// TwinCAT 3 PLC project XTS_PLC
// ProgramVersion: 3.1.4023.0
// libraries:
//   CmpBitmapPool, * (System)
//   Tc2_Math, * (Beckhoff Automation GmbH)
//   Tc2_MC2, * (Beckhoff Automation GmbH)
//   Tc2_Standard, * (Beckhoff Automation GmbH)
//   Tc2_System, * (Beckhoff Automation GmbH)
//   Tc2_Utilities, * (Beckhoff Automation GmbH)
//   Tc3_Mc3Definitions, * (Beckhoff Automation GmbH)
//   Tc3_McCollisionAvoidance, * (Beckhoff Automation GmbH)
//   Tc3_McCoordinatedMotion, * (Beckhoff Automation GmbH)
//   Tc3_Module, * (Beckhoff Automation GmbH)
//   Tc3_XTS_Utility, * (Beckhoff Automation GmbH)
//   VisuDialogs, * (System)
// project tree:
//   DUTs/ eColors.TcDUT, stFeedback.TcDUT, stStationCfg.TcDUT, stTableStructx10.TcDUT, stXTSCfg.TcDUT
//   / GlobalTextList.TcGTLO, PlcTask.TcTTO (not stored), VisualizationManager.TcVMO (not stored)
//   POUs/ MAIN.TcPOU, XTS_PRG.TcPOU
//   POUs/XTS/Group CA/ FB_GroupCA.TcPOU, VI_GroupCAVisu.TcVIS
//   POUs/XTS/Movers/ FB_Mover.TcPOU, FB_MoversFIFO.TcPOU (not stored), MC_JogCA.TcPOU, MC_MoveAbsoluteTimeCA.TcPOU, VI_MoverVisu.TcVIS, VI_MoversVisu.TcVIS
//   POUs/XTS/Stations/ FB_Station.TcPOU, VI_StationVISU.TcVIS, VI_StationsVISU.TcVIS
//   POUs/XTS/VISUs/ GlobalTextList_2.TcGTLO (not stored), VI_PLCOpenState.TcVIS, VI_XTSManualVisu.TcVIS, VI_XTSMainVisu.TcVIS, VI_XTSRunTimeVisu.TcVIS, VI_XTSConfigurationVisu.TcVIS, VI_XTSAutoVisu.TcVIS
//   POUs/XTS/VISUs/TextList/ AxisState_txt.TcTLO, GroupState_txt.TcTLO, MoverMode_TXT.TcTLO (not stored), MoversMode_txt.TcTLO, PML_Modes_txt.TcTLO, StationAckMode_txt.TcTLO (not stored)
//   POUs/XTS/ XTS_System.TcPOU
//   VISUs/ ImagePool.TcIPO (not stored), MAIN_VISU.TcVIS
// real-time tasks:
//   TASK XTS Task 1: cycle T#250us, priority 1, ADS port 350
//   TASK PlcTask: cycle T#10ms, priority 20, ADS port 351
//   TASK VISU_TASK: cycle T#50000us, priority 30, ADS port 352
//   TASK Job Task: cycle default, priority 32
//   TASK VISU_TASK1: cycle T#200000us, priority 2, ADS port 353
// motion (NC):
//   TASK NC-Task 1 SAF: cycle T#2ms, priority 4, ADS port 501
//   TASK NC-Task 1 SVB: cycle T#10ms, priority 8, ADS port 511
//   AXIS Mover Axis 1 (id 1)
//     Dynamic: AccelerationMaximum=80000, DecelerationMaximum=80000, Acceleration=20000, Deceleration=20000, Jerk=200000
//     Velo: Maximum=4000
//     PositionAreaControl: Enable=false
//     TargetPosControl: Enable=false
//     OtherSettings: AllowMotionCmdToSlave=true, AllowMotionCmdToExtSetGenAxis=true
//     encoder EncType=28
//       EncPara: ModuloFactor=10000, ToleranceWndModuloStart=0.2, Inverse=true, MaxCount=#xffffffff
//     drive DrvType=22
//       DrvPara: MaxCount=#xffffffff, DriveControlDWord=#x00000100
//         Analog: VeloReferenz=4200, TorqueSetpointScale=10
//         TimeComp: TaskDelayCycles=1
//     controller CtrType=1
//       CtrPara: PriorControlFactor=1
//         PosDiffControl: Range=10
//         Observer: BandWidth=20
//   AXIS Mover Axis 2 (id 2)
//     Dynamic: AccelerationMaximum=80000, DecelerationMaximum=80000, Acceleration=20000, Deceleration=20000, Jerk=200000
//     Velo: Maximum=4000
//     PositionAreaControl: Enable=false
//     TargetPosControl: Enable=false
//     OtherSettings: AllowMotionCmdToSlave=true, AllowMotionCmdToExtSetGenAxis=true
//     encoder EncType=28
//       EncPara: ModuloFactor=10000, ToleranceWndModuloStart=0.2, MaxCount=#xffffffff
//     drive DrvType=22
//       DrvPara: MaxCount=#xffffffff, DriveControlDWord=#x00000100
//         Analog: VeloReferenz=4200, TorqueSetpointScale=10
//         TimeComp: TaskDelayCycles=1
//     controller CtrType=1
//       CtrPara: PriorControlFactor=1
//         PosDiffControl: Range=10
//         Observer: BandWidth=20
//   AXIS Mover Axis 3 (id 3)
//     Dynamic: AccelerationMaximum=80000, DecelerationMaximum=80000, Acceleration=20000, Deceleration=20000, Jerk=200000
//     Velo: Maximum=4000
//     PositionAreaControl: Enable=false
//     TargetPosControl: Enable=false
//     OtherSettings: AllowMotionCmdToSlave=true, AllowMotionCmdToExtSetGenAxis=true
//     encoder EncType=28
//       EncPara: ModuloFactor=10000, ToleranceWndModuloStart=0.2, MaxCount=#xffffffff
//     drive DrvType=22
//       DrvPara: MaxCount=#xffffffff, DriveControlDWord=#x00000100
//         Analog: VeloReferenz=4200, TorqueSetpointScale=10
//         TimeComp: TaskDelayCycles=1
//     controller CtrType=1
//       CtrPara: PriorControlFactor=1
//         PosDiffControl: Range=10
//         Observer: BandWidth=20
//   AXIS Mover Axis 4 (id 4)
//     Dynamic: AccelerationMaximum=80000, DecelerationMaximum=80000, Acceleration=20000, Deceleration=20000, Jerk=200000
//     Velo: Maximum=4000
//     PositionAreaControl: Enable=false
//     TargetPosControl: Enable=false
//     OtherSettings: AllowMotionCmdToSlave=true, AllowMotionCmdToExtSetGenAxis=true
//     encoder EncType=28
//       EncPara: ModuloFactor=10000, ToleranceWndModuloStart=0.2, MaxCount=#xffffffff
//     drive DrvType=22
//       DrvPara: MaxCount=#xffffffff, DriveControlDWord=#x00000100
//         Analog: VeloReferenz=4200, TorqueSetpointScale=10
//         TimeComp: TaskDelayCycles=1
//     controller CtrType=1
//       CtrPara: PriorControlFactor=1
//         PosDiffControl: Range=10
//         Observer: BandWidth=20
//   AXIS Mover Axis 5 (id 5)
//   AXIS Mover Axis 6 (id 6)
//     Dynamic: AccelerationMaximum=80000, DecelerationMaximum=80000, Acceleration=20000, Deceleration=20000, Jerk=200000
//     Velo: Maximum=4000
//     PositionAreaControl: Enable=false
//     TargetPosControl: Enable=false
//     OtherSettings: AllowMotionCmdToSlave=true, AllowMotionCmdToExtSetGenAxis=true
//     encoder EncType=28
//       EncPara: ModuloFactor=10000, ToleranceWndModuloStart=0.2, MaxCount=#xffffffff
//     drive DrvType=22
//       DrvPara: MaxCount=#xffffffff, DriveControlDWord=#x00000100
//         Analog: VeloReferenz=4200, TorqueSetpointScale=10
//         TimeComp: TaskDelayCycles=1
//     controller CtrType=1
//       CtrPara: PriorControlFactor=1
//         PosDiffControl: Range=10
//         Observer: BandWidth=20
//   AXIS Mover Axis 7 (id 7)
//     Dynamic: AccelerationMaximum=80000, DecelerationMaximum=80000, Acceleration=20000, Deceleration=20000, Jerk=200000
//     Velo: Maximum=4000
//     PositionAreaControl: Enable=false
//     TargetPosControl: Enable=false
//     OtherSettings: AllowMotionCmdToSlave=true, AllowMotionCmdToExtSetGenAxis=true
//     encoder EncType=28
//       EncPara: ModuloFactor=10000, ToleranceWndModuloStart=0.2, MaxCount=#xffffffff
//     drive DrvType=22
//       DrvPara: MaxCount=#xffffffff, DriveControlDWord=#x00000100
//         Analog: VeloReferenz=4200, TorqueSetpointScale=10
//         TimeComp: TaskDelayCycles=1
//     controller CtrType=1
//       CtrPara: PriorControlFactor=1
//         PosDiffControl: Range=10
//         Observer: BandWidth=20
//   AXIS Mover Axis 8 (id 8)
//     Dynamic: AccelerationMaximum=80000, DecelerationMaximum=80000, Acceleration=20000, Deceleration=20000, Jerk=200000
//     Velo: Maximum=4000
//     PositionAreaControl: Enable=false
//     TargetPosControl: Enable=false
//     OtherSettings: AllowMotionCmdToSlave=true, AllowMotionCmdToExtSetGenAxis=true
//     encoder EncType=28
//       EncPara: ModuloFactor=10000, ToleranceWndModuloStart=0.2, MaxCount=#xffffffff
//     drive DrvType=22
//       DrvPara: MaxCount=#xffffffff, DriveControlDWord=#x00000100
//         Analog: VeloReferenz=4200, TorqueSetpointScale=10
//         TimeComp: TaskDelayCycles=1
//     controller CtrType=1
//       CtrPara: PriorControlFactor=1
//         PosDiffControl: Range=10
//         Observer: BandWidth=20
//   AXIS Mover Axis 9 (id 9)
//   AXIS Mover Axis 10 (id 10)
//   AXIS Mover Axis 11 (id 11)
//     Dynamic: AccelerationMaximum=80000, DecelerationMaximum=80000, Acceleration=20000, Deceleration=20000, Jerk=200000
//     Velo: Maximum=4000
//     PositionAreaControl: Enable=false
//     TargetPosControl: Enable=false
//     OtherSettings: AllowMotionCmdToSlave=true, AllowMotionCmdToExtSetGenAxis=true
//     encoder EncType=28
//       EncPara: ModuloFactor=10000, ToleranceWndModuloStart=0.2, MaxCount=#xffffffff
//     drive DrvType=22
//       DrvPara: MaxCount=#xffffffff, DriveControlDWord=#x00000100
//         Analog: VeloReferenz=4200, TorqueSetpointScale=10
//         TimeComp: TaskDelayCycles=1
//     controller CtrType=1
//       CtrPara: PriorControlFactor=1
//         PosDiffControl: Range=10
//         Observer: BandWidth=20
//   AXIS Mover Axis 12 (id 12)
//     Dynamic: AccelerationMaximum=80000, DecelerationMaximum=80000, Acceleration=20000, Deceleration=20000, Jerk=200000
//     Velo: Maximum=4000
//     PositionAreaControl: Enable=false
//     TargetPosControl: Enable=false
//     OtherSettings: AllowMotionCmdToSlave=true, AllowMotionCmdToExtSetGenAxis=true
//     encoder EncType=28
//       EncPara: ModuloFactor=10000, ToleranceWndModuloStart=0.2, MaxCount=#xffffffff
//     drive DrvType=22
//       DrvPara: MaxCount=#xffffffff, DriveControlDWord=#x00000100
//         Analog: VeloReferenz=4200, TorqueSetpointScale=10
//         TimeComp: TaskDelayCycles=1
//     controller CtrType=1
//       CtrPara: PriorControlFactor=1
//         PosDiffControl: Range=10
//         Observer: BandWidth=20
//   AXIS Mover Axis 13 (id 13)
//   AXIS Mover Axis 14 (id 14)
//   AXIS Mover Axis 15 (id 15)
//     Dynamic: AccelerationMaximum=80000, DecelerationMaximum=80000, Acceleration=20000, Deceleration=20000, Jerk=200000
//     Velo: Maximum=4000
//     PositionAreaControl: Enable=false
//     TargetPosControl: Enable=false
//     OtherSettings: AllowMotionCmdToSlave=true, AllowMotionCmdToExtSetGenAxis=true
//     encoder EncType=28
//       EncPara: ModuloFactor=10000, ToleranceWndModuloStart=0.2, MaxCount=#xffffffff
//     drive DrvType=22
//       DrvPara: MaxCount=#xffffffff, DriveControlDWord=#x00000100
//         Analog: VeloReferenz=4200, TorqueSetpointScale=10
//         TimeComp: TaskDelayCycles=1
//     controller CtrType=1
//       CtrPara: PriorControlFactor=1
//         PosDiffControl: Range=10
//         Observer: BandWidth=20
//   AXIS Mover Axis 16 (id 16)
//     Dynamic: AccelerationMaximum=80000, DecelerationMaximum=80000, Acceleration=20000, Deceleration=20000, Jerk=200000
//     Velo: Maximum=4000
//     PositionAreaControl: Enable=false
//     TargetPosControl: Enable=false
//     OtherSettings: AllowMotionCmdToSlave=true, AllowMotionCmdToExtSetGenAxis=true
//     encoder EncType=28
//       EncPara: ModuloFactor=10000, ToleranceWndModuloStart=0.2, MaxCount=#xffffffff
//     drive DrvType=22
//       DrvPara: MaxCount=#xffffffff, DriveControlDWord=#x00000100
//         Analog: VeloReferenz=4200, TorqueSetpointScale=10
//         TimeComp: TaskDelayCycles=1
//     controller CtrType=1
//       CtrPara: PriorControlFactor=1
//         PosDiffControl: Range=10
//         Observer: BandWidth=20
//   AXIS Mover Axis 17 (id 17)
//     Dynamic: AccelerationMaximum=80000, DecelerationMaximum=80000, Acceleration=20000, Deceleration=20000, Jerk=200000
//     Velo: Maximum=4000
//     PositionAreaControl: Enable=false
//     TargetPosControl: Enable=false
//     OtherSettings: AllowMotionCmdToSlave=true, AllowMotionCmdToExtSetGenAxis=true
//     encoder EncType=28
//       EncPara: ModuloFactor=10000, ToleranceWndModuloStart=0.2, MaxCount=#xffffffff
//     drive DrvType=22
//       DrvPara: MaxCount=#xffffffff, DriveControlDWord=#x00000100
//         Analog: VeloReferenz=4200, TorqueSetpointScale=10
//         TimeComp: TaskDelayCycles=1
//     controller CtrType=1
//       CtrPara: PriorControlFactor=1
//         PosDiffControl: Range=10
//         Observer: BandWidth=20
//   AXIS Mover Axis 18 (id 18)
//     General: UnitFlags=#x00000004
//     Dynamic: AccelerationMaximum=80000, DecelerationMaximum=80000, Acceleration=20000, Deceleration=20000, Jerk=200000
//     Velo: Maximum=4000
//     PositionAreaControl: Enable=false
//     TargetPosControl: Enable=false
//     OtherSettings: AllowMotionCmdToSlave=true, AllowMotionCmdToExtSetGenAxis=true
//     encoder EncType=28
//       EncPara: ModuloFactor=10000, ToleranceWndModuloStart=0.2, MaxCount=#xffffffff
//     drive DrvType=22
//       DrvPara: MaxCount=#xffffffff, DriveControlDWord=#x00000100
//         Analog: VeloReferenz=4200, TorqueSetpointScale=10
//         TimeComp: TaskDelayCycles=1
//     controller CtrType=1
//       CtrPara: PriorControlFactor=1
//         PosDiffControl: Range=10
//         Observer: BandWidth=20
//   AXIS Mover Axis 19 (id 19)
//   AXIS Mover Axis 20 (id 20)
//     Dynamic: AccelerationMaximum=80000, DecelerationMaximum=80000, Acceleration=20000, Deceleration=20000, Jerk=200000
//     Velo: Maximum=4000
//     PositionAreaControl: Enable=false
//     TargetPosControl: Enable=false
//     OtherSettings: AllowMotionCmdToSlave=true, AllowMotionCmdToExtSetGenAxis=true
//     encoder EncType=28
//       EncPara: ModuloFactor=10000, ToleranceWndModuloStart=0.2, MaxCount=#xffffffff
//     drive DrvType=22
//       DrvPara: MaxCount=#xffffffff, DriveControlDWord=#x00000100
//         Analog: VeloReferenz=4200, TorqueSetpointScale=10
//         TimeComp: TaskDelayCycles=1
//     controller CtrType=1
//       CtrPara: PriorControlFactor=1
//         PosDiffControl: Range=10
//         Observer: BandWidth=20
//   AXIS Mover Axis 21 (id 21)
// I/O:
//   DEVICE Device 3
//   DEVICE Device 2 (EtherCAT) (disabled), AmsNetId 10.55.2.47.3.1
// variable links:
//   (this object) <-> TcCOM Objects/XtsProcessingUnit 1/Mover 1
//     SoftDrive 1/Data Pointer/InputPointer1 <-> Inputs/SoftDriveInput
//     SoftDrive 1/Data Pointer/OutputPointer1 <-> Outputs/SoftDriveOutput
//   (this object) <-> TcCOM Objects/XtsProcessingUnit 1/Mover 2
//     SoftDrive 2/Data Pointer/InputPointer1 <-> Inputs/SoftDriveInput
//     SoftDrive 2/Data Pointer/OutputPointer1 <-> Outputs/SoftDriveOutput
//   (this object) <-> TcCOM Objects/XtsProcessingUnit 1/Mover 3
//     SoftDrive 3/Data Pointer/InputPointer1 <-> Inputs/SoftDriveInput
//     SoftDrive 3/Data Pointer/OutputPointer1 <-> Outputs/SoftDriveOutput
//   (this object) <-> TcCOM Objects/XtsProcessingUnit 1/Mover 4
//     SoftDrive 4/Data Pointer/InputPointer1 <-> Inputs/SoftDriveInput
//     SoftDrive 4/Data Pointer/OutputPointer1 <-> Outputs/SoftDriveOutput
//   (this object) <-> TcCOM Objects/XtsProcessingUnit 1/Mover 6
//     SoftDrive 6/Data Pointer/InputPointer1 <-> Inputs/SoftDriveInput
//     SoftDrive 6/Data Pointer/OutputPointer1 <-> Outputs/SoftDriveOutput
//   (this object) <-> TcCOM Objects/XtsProcessingUnit 1/Mover 7
//     SoftDrive 7/Data Pointer/InputPointer1 <-> Inputs/SoftDriveInput
//     SoftDrive 7/Data Pointer/OutputPointer1 <-> Outputs/SoftDriveOutput
//   (this object) <-> TcCOM Objects/XtsProcessingUnit 1/Mover 8
//     SoftDrive 8/Data Pointer/InputPointer1 <-> Inputs/SoftDriveInput
//     SoftDrive 8/Data Pointer/OutputPointer1 <-> Outputs/SoftDriveOutput
//   (this object) <-> TcCOM Objects/XtsProcessingUnit 1/Mover 11
//     SoftDrive 11/Data Pointer/InputPointer1 <-> Inputs/SoftDriveInput
//     SoftDrive 11/Data Pointer/OutputPointer1 <-> Outputs/SoftDriveOutput
//   (this object) <-> TcCOM Objects/XtsProcessingUnit 1/Mover 12
//     SoftDrive 12/Data Pointer/InputPointer1 <-> Inputs/SoftDriveInput
//     SoftDrive 12/Data Pointer/OutputPointer1 <-> Outputs/SoftDriveOutput
//   (this object) <-> TcCOM Objects/XtsProcessingUnit 1/Mover 15
//     SoftDrive 15/Data Pointer/InputPointer1 <-> Inputs/SoftDriveInput
//     SoftDrive 15/Data Pointer/OutputPointer1 <-> Outputs/SoftDriveOutput
//   (this object) <-> TcCOM Objects/XtsProcessingUnit 1/Mover 16
//     SoftDrive 16/Data Pointer/InputPointer1 <-> Inputs/SoftDriveInput
//     SoftDrive 16/Data Pointer/OutputPointer1 <-> Outputs/SoftDriveOutput
//   (this object) <-> TcCOM Objects/XtsProcessingUnit 1/Mover 17
//     SoftDrive 17/Data Pointer/InputPointer1 <-> Inputs/SoftDriveInput
//     SoftDrive 17/Data Pointer/OutputPointer1 <-> Outputs/SoftDriveOutput
//   (this object) <-> TcCOM Objects/XtsProcessingUnit 1/Mover 18
//     SoftDrive 18/Data Pointer/InputPointer1 <-> Inputs/SoftDriveInput
//     SoftDrive 18/Data Pointer/OutputPointer1 <-> Outputs/SoftDriveOutput
//   (this object) <-> TcCOM Objects/XtsProcessingUnit 1/Mover 20
//     SoftDrive 20/Data Pointer/InputPointer1 <-> Inputs/SoftDriveInput
//     SoftDrive 20/Data Pointer/OutputPointer1 <-> Outputs/SoftDriveOutput
//   XTS_PLC Instance <-> NC-Task 1 SAF/Axes/Mover Axis 1
//     PlcTask Inputs/XTS_PRG.fbXTSSystem.ax[1].ax.NcToPlc <-> Outputs/ToPlc
//     PlcTask Outputs/XTS_PRG.fbXTSSystem.ax[1].ax.PlcToNc <-> Inputs/FromPlc
//   XTS_PLC Instance <-> NC-Task 1 SAF/Axes/Mover Axis 10
//     PlcTask Inputs/XTS_PRG.fbXTSSystem.ax[10].ax.NcToPlc <-> Outputs/ToPlc
//     PlcTask Outputs/XTS_PRG.fbXTSSystem.ax[10].ax.PlcToNc <-> Inputs/FromPlc
//   XTS_PLC Instance <-> NC-Task 1 SAF/Axes/Mover Axis 11
//     PlcTask Inputs/XTS_PRG.fbXTSSystem.ax[11].ax.NcToPlc <-> Outputs/ToPlc
//     PlcTask Outputs/XTS_PRG.fbXTSSystem.ax[11].ax.PlcToNc <-> Inputs/FromPlc
//   XTS_PLC Instance <-> NC-Task 1 SAF/Axes/Mover Axis 12
//     PlcTask Inputs/XTS_PRG.fbXTSSystem.ax[12].ax.NcToPlc <-> Outputs/ToPlc
//     PlcTask Outputs/XTS_PRG.fbXTSSystem.ax[12].ax.PlcToNc <-> Inputs/FromPlc
//   XTS_PLC Instance <-> NC-Task 1 SAF/Axes/Mover Axis 13
//     PlcTask Inputs/XTS_PRG.fbXTSSystem.ax[13].ax.NcToPlc <-> Outputs/ToPlc
//     PlcTask Outputs/XTS_PRG.fbXTSSystem.ax[13].ax.PlcToNc <-> Inputs/FromPlc
//   XTS_PLC Instance <-> NC-Task 1 SAF/Axes/Mover Axis 14
//     PlcTask Inputs/XTS_PRG.fbXTSSystem.ax[14].ax.NcToPlc <-> Outputs/ToPlc
//     PlcTask Outputs/XTS_PRG.fbXTSSystem.ax[14].ax.PlcToNc <-> Inputs/FromPlc
//   XTS_PLC Instance <-> NC-Task 1 SAF/Axes/Mover Axis 15
//     PlcTask Inputs/XTS_PRG.fbXTSSystem.ax[15].ax.NcToPlc <-> Outputs/ToPlc
//     PlcTask Outputs/XTS_PRG.fbXTSSystem.ax[15].ax.PlcToNc <-> Inputs/FromPlc
//   XTS_PLC Instance <-> NC-Task 1 SAF/Axes/Mover Axis 16
//     PlcTask Inputs/XTS_PRG.fbXTSSystem.ax[16].ax.NcToPlc <-> Outputs/ToPlc
//     PlcTask Outputs/XTS_PRG.fbXTSSystem.ax[16].ax.PlcToNc <-> Inputs/FromPlc
//   XTS_PLC Instance <-> NC-Task 1 SAF/Axes/Mover Axis 17
//     PlcTask Inputs/XTS_PRG.fbXTSSystem.ax[17].ax.NcToPlc <-> Outputs/ToPlc
//     PlcTask Outputs/XTS_PRG.fbXTSSystem.ax[17].ax.PlcToNc <-> Inputs/FromPlc
//   XTS_PLC Instance <-> NC-Task 1 SAF/Axes/Mover Axis 18
//     PlcTask Inputs/XTS_PRG.fbXTSSystem.ax[18].ax.NcToPlc <-> Outputs/ToPlc
//     PlcTask Outputs/XTS_PRG.fbXTSSystem.ax[18].ax.PlcToNc <-> Inputs/FromPlc
//   XTS_PLC Instance <-> NC-Task 1 SAF/Axes/Mover Axis 19
//     PlcTask Inputs/XTS_PRG.fbXTSSystem.ax[19].ax.NcToPlc <-> Outputs/ToPlc
//     PlcTask Outputs/XTS_PRG.fbXTSSystem.ax[19].ax.PlcToNc <-> Inputs/FromPlc
//   XTS_PLC Instance <-> NC-Task 1 SAF/Axes/Mover Axis 2
//     PlcTask Inputs/XTS_PRG.fbXTSSystem.ax[2].ax.NcToPlc <-> Outputs/ToPlc
//     PlcTask Outputs/XTS_PRG.fbXTSSystem.ax[2].ax.PlcToNc <-> Inputs/FromPlc
//   XTS_PLC Instance <-> NC-Task 1 SAF/Axes/Mover Axis 20
//     PlcTask Inputs/XTS_PRG.fbXTSSystem.ax[20].ax.NcToPlc <-> Outputs/ToPlc
//     PlcTask Outputs/XTS_PRG.fbXTSSystem.ax[20].ax.PlcToNc <-> Inputs/FromPlc
//   XTS_PLC Instance <-> NC-Task 1 SAF/Axes/Mover Axis 21
//     PlcTask Inputs/XTS_PRG.fbXTSSystem.ax[21].ax.NcToPlc <-> Outputs/ToPlc
//     PlcTask Outputs/XTS_PRG.fbXTSSystem.ax[21].ax.PlcToNc <-> Inputs/FromPlc
//   XTS_PLC Instance <-> NC-Task 1 SAF/Axes/Mover Axis 3
//     PlcTask Inputs/XTS_PRG.fbXTSSystem.ax[3].ax.NcToPlc <-> Outputs/ToPlc
//     PlcTask Outputs/XTS_PRG.fbXTSSystem.ax[3].ax.PlcToNc <-> Inputs/FromPlc
//   XTS_PLC Instance <-> NC-Task 1 SAF/Axes/Mover Axis 4
//     PlcTask Inputs/XTS_PRG.fbXTSSystem.ax[4].ax.NcToPlc <-> Outputs/ToPlc
//     PlcTask Outputs/XTS_PRG.fbXTSSystem.ax[4].ax.PlcToNc <-> Inputs/FromPlc
//   XTS_PLC Instance <-> NC-Task 1 SAF/Axes/Mover Axis 5
//     PlcTask Inputs/XTS_PRG.fbXTSSystem.ax[5].ax.NcToPlc <-> Outputs/ToPlc
//     PlcTask Outputs/XTS_PRG.fbXTSSystem.ax[5].ax.PlcToNc <-> Inputs/FromPlc
//   XTS_PLC Instance <-> NC-Task 1 SAF/Axes/Mover Axis 6
//     PlcTask Inputs/XTS_PRG.fbXTSSystem.ax[6].ax.NcToPlc <-> Outputs/ToPlc
//     PlcTask Outputs/XTS_PRG.fbXTSSystem.ax[6].ax.PlcToNc <-> Inputs/FromPlc
//   XTS_PLC Instance <-> NC-Task 1 SAF/Axes/Mover Axis 7
//     PlcTask Inputs/XTS_PRG.fbXTSSystem.ax[7].ax.NcToPlc <-> Outputs/ToPlc
//     PlcTask Outputs/XTS_PRG.fbXTSSystem.ax[7].ax.PlcToNc <-> Inputs/FromPlc
//   XTS_PLC Instance <-> NC-Task 1 SAF/Axes/Mover Axis 8
//     PlcTask Inputs/XTS_PRG.fbXTSSystem.ax[8].ax.NcToPlc <-> Outputs/ToPlc
//     PlcTask Outputs/XTS_PRG.fbXTSSystem.ax[8].ax.PlcToNc <-> Inputs/FromPlc
//   XTS_PLC Instance <-> NC-Task 1 SAF/Axes/Mover Axis 9
//     PlcTask Inputs/XTS_PRG.fbXTSSystem.ax[9].ax.NcToPlc <-> Outputs/ToPlc
//     PlcTask Outputs/XTS_PRG.fbXTSSystem.ax[9].ax.PlcToNc <-> Inputs/FromPlc
//   XTS_PLC Instance <-> NC-Task 1 SAF/Objects/Group1 (CA Group)
//     PlcTask Inputs/XTS_PRG.fbXTSSystem.gp.ag.NcToPlc <-> Group Outputs/ToPLC
//     PlcTask Outputs/XTS_PRG.fbXTSSystem.gp.ag.PlcToNc <-> Group Inputs/FromPLC

// ---- DUTs/eColors.TcDUT
{attribute 'qualified_only'}
{attribute 'strict'}
TYPE eColors :
(
	red := 16#FFFF0000,
	green := 16#FF00FF00,
	blue := 16#FF0000FF,
	orange := 16#FFFF8000
)DWORD;
END_TYPE

// ---- DUTs/stFeedback.TcDUT
TYPE stFeedback :
STRUCT
	bBusy			: BOOL;
	bDone			: BOOL;
	bCommandAborted : BOOL;
	bError			: BOOL;
	udiErrorID		: UDINT;
END_STRUCT
END_TYPE

// ---- DUTs/stStationCfg.TcDUT
TYPE stStationCfg :
STRUCT
	sName					: STRING;
	lrStartPosition			: LREAL;
	lrEndPosition			: LREAL;
	lrStopPosition			: ARRAY [1..3] OF LREAL;
	lrProcessingTime		: LREAL;
	uiNumStopPositions		: UDINT;
	lrTravelTime			: LREAL;
	bEnableManualAck		: BOOL;
	bManualAck				: BOOL;
END_STRUCT
END_TYPE

// ---- DUTs/stTableStructx10.TcDUT
TYPE stTableStructx10 :
STRUCT
	b1 : BOOL;
		b2 : BOOL;
			b3 : BOOL;
				b4 : BOOL;
					b5 : BOOL;
						b6 : BOOL;
							b7 : BOOL;
								b8 : BOOL;
									b9 : BOOL;
										b10 : BOOL;
END_STRUCT
END_TYPE

// ---- DUTs/stXTSCfg.TcDUT
TYPE stXTSCfg :
STRUCT
	bInvertPolarity			: BOOL;
	udiNumStations			: UDINT;
	udiMoverMode			: UDINT := 1; //1 --> Single, 2 --> Double, 3 --> Triple
	lrMoverDistance			: LREAL := 60.0; //Distance between movers when Mover mode is different of single
	stStationsCfg 			: ARRAY [1..Tc3_XTS_Utility.TcIoXtsEnvironmentParameterList.MaxXtsInfoStation] OF stStationCfg;
	bNotCfgStationsViewer	: BOOL := FALSE;
END_STRUCT
END_TYPE

// ---- POUs/MAIN.TcPOU
PROGRAM MAIN


//XTS Program Call
XTS_PRG();

END_PROGRAM

// ---- POUs/XTS_PRG.TcPOU
PROGRAM XTS_PRG
VAR
	fbXTSSystem : XTS_System;
	bInit		: BOOL := FALSE;
	i			: UDINT;
END_VAR

IF bInit = FALSE THEN
		
		fbXTSSystem.stCfg.udiMoverMode							:= 1; //Single
		fbXTSSystem.stCfg.bInvertPolarity						:= FALSE;

		fbXTSSystem.stCfg.udiNumStations						:= 3;
		fbXTSSystem.stCfg.stStationsCfg[1].sName			 	:= 'Station 1'; 
		fbXTSSystem.stCfg.stStationsCfg[1].lrStartPosition 		:= 0.0; 
		fbXTSSystem.stCfg.stStationsCfg[1].lrEndPosition	 	:= 500.0; 
		fbXTSSystem.stCfg.stStationsCfg[1].lrStopPosition[1] 	:= 100.0; 
		fbXTSSystem.stCfg.stStationsCfg[1].lrStopPosition[2] 	:= 450.0; 
		fbXTSSystem.stCfg.stStationsCfg[1].lrProcessingTime 	:= 1.0;
		fbXTSSystem.stCfg.stStationsCfg[1].uiNumStopPositions 	:= 1;
		fbXTSSystem.stCfg.stStationsCfg[1].lrTravelTime			:= 0.5;				

		fbXTSSystem.stCfg.stStationsCfg[2].sName			 	:= 'Station 2'; 		
		fbXTSSystem.stCfg.stStationsCfg[2].lrStartPosition 		:= 1000.0; 
		fbXTSSystem.stCfg.stStationsCfg[2].lrEndPosition	 	:= 1500.0;
		fbXTSSystem.stCfg.stStationsCfg[2].lrStopPosition[1]	:= 10.0; 
		fbXTSSystem.stCfg.stStationsCfg[2].lrStopPosition[2]	:= 250.0; 
		fbXTSSystem.stCfg.stStationsCfg[2].lrStopPosition[3]	:= 500.0; 
		fbXTSSystem.stCfg.stStationsCfg[2].lrProcessingTime 	:= 3.0;
		fbXTSSystem.stCfg.stStationsCfg[2].uiNumStopPositions 	:= 3;
		fbXTSSystem.stCfg.stStationsCfg[2].lrTravelTime			:= 0.5;				

 		fbXTSSystem.stCfg.stStationsCfg[3].sName			 	:= 'Station 3';  
		fbXTSSystem.stCfg.stStationsCfg[3].lrStartPosition 		:= 2000.0; 
		fbXTSSystem.stCfg.stStationsCfg[3].lrEndPosition	 	:= 2500.0;
		fbXTSSystem.stCfg.stStationsCfg[3].lrStopPosition[1] 	:= 100.0; 
		fbXTSSystem.stCfg.stStationsCfg[3].lrProcessingTime 	:= 1.0;
		fbXTSSystem.stCfg.stStationsCfg[3].uiNumStopPositions 	:= 1;
		fbXTSSystem.stCfg.stStationsCfg[3].lrTravelTime			:= 0.5;				

		fbXTSSystem.stCfg.stStationsCfg[4].sName			 	:= 'Station 4'; 	
		fbXTSSystem.stCfg.stStationsCfg[4].lrStartPosition 		:= 3000.0; 
		fbXTSSystem.stCfg.stStationsCfg[4].lrEndPosition	 	:= 3500.0;
		fbXTSSystem.stCfg.stStationsCfg[4].lrStopPosition[1] 	:= 200.0; 
		fbXTSSystem.stCfg.stStationsCfg[4].lrProcessingTime 	:= 1.0;
		fbXTSSystem.stCfg.stStationsCfg[4].uiNumStopPositions 	:= 1;
		fbXTSSystem.stCfg.stStationsCfg[4].lrTravelTime			:= 0.5;				

		fbXTSSystem.stCfg.stStationsCfg[5].sName			 	:= 'Station 5'; 
		fbXTSSystem.stCfg.stStationsCfg[5].lrStartPosition 		:= 4000.0; 
		fbXTSSystem.stCfg.stStationsCfg[5].lrEndPosition	 	:= 4500.0;
		fbXTSSystem.stCfg.stStationsCfg[5].lrStopPosition[1] 	:= 300.0; 
		fbXTSSystem.stCfg.stStationsCfg[5].lrProcessingTime 	:= 1.0;
		fbXTSSystem.stCfg.stStationsCfg[5].uiNumStopPositions 	:= 1;
		fbXTSSystem.stCfg.stStationsCfg[5].lrTravelTime			:= 0.5;				

		fbXTSSystem.stCfg.stStationsCfg[6].sName			 	:= 'Station 6'; 
		fbXTSSystem.stCfg.stStationsCfg[6].lrStartPosition 		:= 5000.0; 
		fbXTSSystem.stCfg.stStationsCfg[6].lrEndPosition	 	:= 5500.0;
		fbXTSSystem.stCfg.stStationsCfg[6].lrStopPosition[1] 	:= 25.0; 
		fbXTSSystem.stCfg.stStationsCfg[6].lrStopPosition[2] 	:= 325.0; 
		fbXTSSystem.stCfg.stStationsCfg[6].lrStopPosition[3] 	:= 500.0; 
		fbXTSSystem.stCfg.stStationsCfg[6].lrProcessingTime 	:= 3.0;
		fbXTSSystem.stCfg.stStationsCfg[6].uiNumStopPositions 	:= 2;
		fbXTSSystem.stCfg.stStationsCfg[6].lrTravelTime			:= 0.5;				

		fbXTSSystem.stCfg.stStationsCfg[7].sName			 	:= 'Station 7'; 
		fbXTSSystem.stCfg.stStationsCfg[7].lrStartPosition 		:= 6000.0; 
		fbXTSSystem.stCfg.stStationsCfg[7].lrEndPosition	 	:= 8500.0;	
		fbXTSSystem.stCfg.stStationsCfg[7].lrStopPosition[1] 	:= 10.0; 
		fbXTSSystem.stCfg.stStationsCfg[7].lrStopPosition[2] 	:= 650.0;
		fbXTSSystem.stCfg.stStationsCfg[7].lrStopPosition[3] 	:= 1200.0;
		fbXTSSystem.stCfg.stStationsCfg[7].lrProcessingTime 	:= 3.0;
		fbXTSSystem.stCfg.stStationsCfg[7].uiNumStopPositions 	:= 3;
		fbXTSSystem.stCfg.stStationsCfg[7].lrTravelTime			:= 0.5;
		
		fbXTSSystem.bEnable := TRUE;
		
		FOR i:=1 TO fbXTSSystem.stCfg.udiNumStations DO
			fbXTSSystem.stCfg.stStationsCfg[i].bEnableManualAck	:= FALSE;
		END_FOR

		bInit := TRUE;				
END_IF
fbXTSSystem.cyclic();

END_PROGRAM

// ---- POUs/XTS/XTS_System.TcPOU
FUNCTION_BLOCK XTS_System
VAR_INPUT
{attribute 'pingroup' := 'Power'}
	bEnable					: BOOL := FALSE;	//Enable operation (power movers, group all ...)
{attribute 'pingroup' := 'Power'}
	bReset					: BOOL := FALSE;	//Reset all axis
{attribute 'pingroup' := 'Manual'}
	bManual					: BOOL;				//Manual operation mode for movers test with collision avoidance
{attribute 'pingroup' := 'Manual'}
	udiMoverSelection		: UDINT := 0;		//Mover ID to move in manual mode. If ID is equal to zero all movers are moved
{attribute 'pingroup' := 'Manual'}
	udiStationSelection		: UDINT := 0;		//Target Station ID for mover selected. If zero manual mode works with target position input
{attribute 'pingroup' := 'Manual'}
	udiStopPositionSelection: UDINT := 1;		//Stop position selection 1, 2 or 3
{attribute 'pingroup' := 'Manual'}
	bJogForward				: BOOL;				//Jog Forward command for manual mode operation 0
{attribute 'pingroup' := 'Manual'}
	bJogBackwards			: BOOL;				//Jog Backwards command for manual mode operation 0
{attribute 'pingroup' := 'Manual'}
	bManualMove				: BOOL;				//Move selected mover to target position at target velocity in manual mode operation 1
{attribute 'pingroup' := 'Manual'}
	bTeachStation			: BOOL;				//During manual mode flag up of teach station set the stop position of station equal to act mover position
{attribute 'pingroup' := 'Automatic'}
	bAutomatic				: BOOL;				//Automatic operation using stations
{attribute 'pingroup' := 'Profile'}
	lrTargetPosition		: LREAL := 0.0;		//Target Position [mm]
{attribute 'pingroup' := 'Profile'}
	lrTargetVelocity		: LREAL := 500.0;	//Target Velocity [mm]
{attribute 'pingroup' := 'Configuration'}
	stCfg					: stXTSCfg;			//General Configuration
{attribute 'pingroup' := 'Profile'}
	Direction				: tc3_mc3definitions.MC_DIRECTION := tc3_mc3definitions.MC_DIRECTION.mcDirectionPositive;	//Movement Direction	
{attribute 'pingroup' := 'SubElements'}
	ax						: ARRAY [1..Tc3_XTS_Utility.TcIoXtsEnvironmentParameterList.MaxXtsMoversPerXpu] OF FB_Mover;	//Movers
{attribute 'pingroup' := 'SubElements'}
	gp						: FB_GroupCA; //Group CA
{attribute 'pingroup' := 'SubElements'}
	aStations				: ARRAY [1..Tc3_XTS_Utility.TcIoXtsEnvironmentParameterList.MaxXtsInfoStation] OF FB_Station; //Stations
END_VAR
VAR_OUTPUT
{attribute 'pingroup' := 'Status'}
	sLog			 			: STRING := 'Invalid';
{attribute 'pingroup' := 'Status'}
	bError			 			: BOOL;
{attribute 'pingroup' := 'Status'}
	bReadyForMotion 			: BOOL;
{attribute 'pingroup' := 'Status'}
	bEnabled					: BOOL;
{attribute 'pingroup' := 'Manual'}
	bInManual					: BOOL;
{attribute 'pingroup' := 'Manual'}
	bTeachDone					: BOOL;
{attribute 'pingroup' := 'Automatic'}
	bInAutomatic				: BOOL;
{attribute 'pingroup' := 'XPU'}
	bInitDone					: BOOL;
{attribute 'pingroup' := 'XPU'}
	bMover1DetectionValid 		: BOOL;
{attribute 'pingroup' := 'XPU'}
	iOperationMode 				: OperationMode;
{attribute 'pingroup' := 'XPU'}
	AreAllPositionValid 		: BOOL;
{attribute 'pingroup' := 'XPU'}
	DetectedMoverCount 			: UDINT;
{attribute 'pingroup' := 'XPU'}
	ExpectedMoverCount 			: UDINT;
{attribute 'pingroup' := 'XPU'}
	HasMoverIdDetectorError		: BOOL;
{attribute 'pingroup' := 'XPU'}
	IsMoverIdDetectorActive		: BOOL;
{attribute 'pingroup' := 'XPU'}
	IsMoverIsDetectionValid		: BOOL;
{attribute 'pingroup' := 'XPU'}
	TrackCount					: UDINT;	
{attribute 'pingroup' := 'XPU'}
	PartCount					: UDINT;				
{attribute 'pingroup' := 'XPU'}
	lrPart1Length 				: LREAL;
{attribute 'pingroup' := 'XPU'}
	udiNumMovers  				: UDINT;
{attribute 'pingroup' := 'XPU'}
	udiPart1NumModules			: UDINT;
{attribute 'pingroup' := 'XPU'}
	eMoverType					: Tc3_XTS_Utility.MoverType;
{attribute 'pingroup' := 'GROUP CA'}
	eGroupState					: MC_GROUP_STATE;
{attribute 'pingroup' := 'GROUP CA'}
	bAllMoversStandStill		: BOOL;	
END_VAR
VAR
	(* XPU *)
	//{attribute 'hide'} 
	fbXTSEnv		 		: FB_TcIoXtsEnvironment;
	//{attribute 'hide'} 
	IXPU			 		: I_TcIoXtsProcessingUnit;
	//{attribute 'hide'} 
	IPart1			 		: I_TcIoXtsXpuPart;
	//{attribute 'hide'} 
	fbInfoServer			: FB_TcIoXtsInfoServer;
	//{attribute 'hide'} 
	aInfoServerOids			: ARRAY [1..Tc3_XTS_Utility.TcIoXtsEnvironmentParameterList.MaxXtsInfoServer] OF Tc3_XTS_Utility.OTCID;
	//{attribute 'hide'} 
	aStationsOTCID			: ARRAY [1..Tc3_XTS_Utility.TcIoXtsEnvironmentParameterList.MaxXtsInfoStation] OF Tc3_XTS_Utility.OTCID;
	//{attribute 'hide'} 
	aMoversOids				: ARRAY [1..Tc3_XTS_Utility.TcIoXtsEnvironmentParameterList.MaxXtsMoversPerXpu] OF Tc3_XTS_Utility.OTCID;
	//{attribute 'hide'} 
	GroupCAOTCID			: ARRAY [1..Tc3_XTS_Utility.TcIoXtsEnvironmentParameterList.MaxXtsCaGroup] OF Tc3_XTS_Utility.OTCID;
END_VAR
VAR
	bXPUInitDone			: BOOL;
	stVisuStationsCfg 		: ARRAY [1..Tc3_XTS_Utility.TcIoXtsEnvironmentParameterList.MaxXtsInfoStation] OF stStationCfg;
	stCurrentCfg			: stXTSCfg;			//General Configuration
	udiFirstMover			: UDINT;
END_VAR
VAR
	//Visu
	iFrameSelection				: INT;
	iVisuMoverSelection			: INT := 1;		//Mover ID to move in manual mode. If ID is equal to zero all movers are moved
	iVisuStationSelection		: INT := 1;		//Target Station ID for mover selected. If zero manual mode works with target position input
	iVisuStopPositionSelection	: INT := 2;		//Target Stop Position 1, 2 or 3
END_VAR

METHOD PRIVATE Automatic : BOOL
VAR_INPUT
	bEnable : BOOL;
END_VAR
VAR_INST
	iState 		: INT;
	bAllDone 	: BOOL;
	i 			: UDINT;
	bBusy		: BOOL;
	udiErrorID	: UDINT;
END_VAR

//Error managment
IF (bError OR bReset) AND iState <> 999 AND bBusy = TRUE THEN iState := 999; END_IF

CASE iState OF
	
	0 : IF bEnable THEN 
			stCurrentCfg := stCfg;
			//Reset all command
			FOR i:= 1 TO udiNumMovers DO
				ax[i].clearCmd();
			END_FOR
			iState := iState + 1; 
			bBusy  := TRUE;
		END_IF
		
	1 : //ReConfigure Stations
		sLog := CONCAT('Auto: Configure stations, State: ', INT_TO_STRING(iState));
		IF ConfigureStations() THEN iState := iState + 1; END_IF

	2 : //Put all stations in auto mode
		sLog := CONCAT('Auto: starting Stations secuence, State: ', INT_TO_STRING(iState));
		bAllDOne := TRUE;
		FOR i:= 1 TO stCurrentCfg.udiNumStations DO
			bAllDone := bAllDOne AND aStations[i].Start();
			IF udiErrorID <> 0 THEN
				sLog := '';
				sLog := CONCAT('Auto: Error in station: ', UDINT_TO_STRING(i));
				iState := 1000;		
			END_IF
		END_FOR
		IF bAllDone THEN iState := iState + 1; END_IF
		IF bEnable = FALSE THEN iState := 100; END_IF
		
	3 : //Move all to zero position
		sLog := CONCAT('Auto: Move movers to start position, State: ', INT_TO_STRING(iState));
		bAllDOne := FALSE;
		FOR i:= 1 TO udiNumMovers DO
			IF stCurrentCfg.udiMoverMode <> 1 THEN
				bAllDone := bAllDOne OR ax[i].moveca_gap(TRUE, 0.0, 1000.0, stCurrentCfg.lrMoverDistance).bDone;
			ELSE
				bAllDone := bAllDOne OR ax[i].moveca(TRUE, 0.0, 1000.0).bDone;
			END_IF
		END_FOR
		IF bAllMoversStandStill AND bAllDone THEN
			udiFirstMover := WhoIsAtPos(0.0);
			FOR i:= 1 TO udiNumMovers DO
				ax[i].moveca(FALSE, 0.1, 0.0);
			END_FOR
			IF udiFirstMover <> 0 THEN
				iState := iState + 1;
			END_IF
		END_IF
		IF bEnable = FALSE THEN 
			iState := 100; 
		END_IF
		
	4 : //Gear in passive movers
		sLog := CONCAT('Auto: Gear in passive movers, State: ', INT_TO_STRING(iState));
		bAllDone := TRUE;
		FOR i:= 1 TO udiNumMovers DO
			IF IsPassiveMover(i) THEN
				IF ax[1].bMoverInverted = FALSE THEN 
					bAllDone := bAllDone AND ax[i].gearIn(TRUE, 1, 1, ax[SEL(i = udiNumMovers, i+1, 1)].p_Axis).bDone;
					IF udiErrorID <> 0 THEN
						sLog := '';
						sLog := CONCAT('Auto: Error Gear in axis: ', UDINT_TO_STRING(i));
						iState := 1000;		
					END_IF
				ELSE
					bAllDone := bAllDone AND ax[i].gearIn(TRUE, 1, 1, ax[SEL(i = 1, i-1, udiNumMovers)].p_Axis).bDone;
					IF udiErrorID <> 0 THEN
						sLog := '';
						sLog := CONCAT('Auto: Error Gear in axis: ', UDINT_TO_STRING(i));
						iState := 1000;		
					END_IF
				END_IF
			END_IF
		END_FOR
		IF bAllDone THEN
			FOR i:= 1 TO udiNumMovers DO
				IF IsPassiveMover(i) THEN
					bAllDone := bAllDone AND ax[i].gearIn(FALSE, 1, 1, ax[SEL(i = udiNumMovers, i+1, 1)].p_Axis).bDone;
				END_IF
			END_FOR
			iState := iState + 1;
		END_IF

	5 :  //Add Movers to first station
		sLog := CONCAT('Auto: Add Movers to first station, State: ', INT_TO_STRING(iState)); 
		FOR i:= 1 TO udiNumMovers DO
			IF IsPassiveMover(i) = FALSE THEN
				aStations[1].RegisterMover(ax[i].udiID);				
			END_IF
		END_FOR
		iState := iState + 1;
	
	6 : //Call stations auto mode
		sLog := CONCAT('Auto: Running, State: ', INT_TO_STRING(iState));
		bAllDOne := TRUE;
		(*FOR i:= 1 TO stCurrentCfg.udiNumStations DO
			bAllDone := bAllDOne AND aStations[i].Sequence2(TRUE, FALSE, m_udiErrorID => udiErrorID);
			IF udiErrorID <> 0 THEN
				sLog := '';
				sLog := CONCAT('Auto: Error in station: ', UDINT_TO_STRING(i));
				iState := 1000;		
			END_IF
		END_FOR*)
		IF bEnable = FALSE THEN 
			iState := 100; 
		END_IF
	
	100 : //Stop
		sLog := CONCAT('Auto: Exit stations from auto mode, State: ', INT_TO_STRING(iState));
		bAllDOne := TRUE;
		FOR i:= 1 TO stCurrentCfg.udiNumStations DO
			bAllDone := bAllDOne AND NOT aStations[i].Stop();
		END_FOR
		IF bAllDone THEN
			iState := iState + 1;
		END_IF
		
	101 : //Check for all StandStill
		sLog := CONCAT('Auto: Check all movers at standstill, State: ', INT_TO_STRING(iState));
		bAllDone := TRUE;
		FOR i := 1 TO udiNumMovers DO
			bAllDone := bAllDone AND ax[i].standstill();
		END_FOR
		IF bAllDOne THEN
			iState := iState + 1;
		END_IF
		
	102 : //Gear Out
		sLog := CONCAT('Auto: Gear out, State: ', INT_TO_STRING(iState));
		bAllDone := TRUE;
		FOR i := 1 TO udiNumMovers DO
			IF IsPassiveMover(i) THEN
				bAllDone := bAllDone AND ax[i].gearOut(TRUE).bDone;
			END_IF
		END_FOR
		IF bAllDOne THEN
			FOR i := 1 TO udiNumMovers DO
				IF IsPassiveMover(i) THEN
					ax[i].gearOut(FALSE);
				END_IF
			END_FOR
			iState := iState + 1;
		END_IF
		
	103 : bBusy := FALSE;
		sLog := CONCAT('Auto: End, State: ', INT_TO_STRING(iState));
		IF bEnable = FALSE THEN
			iState := 0;
		END_IF
		
	999 : //Error State 
		bBusy := FALSE;
		sLog := CONCAT('Auto: Abort, State: ', INT_TO_STRING(iState));
		FOR i:=1 TO stCurrentCfg.udiNumStations DO
			//Abort Station Sequence
			aStations[i].Stop();
		END_FOR
		IF bEnable = FALSE THEN
			sLog := CONCAT('Auto: End, State: ', INT_TO_STRING(iState));
			iState := 0;
		END_IF
		
	1000 : //Internal Error
		bBusy := FALSE;
		IF bEnable = FALSE THEN
			FOR i:=1 TO stCurrentCfg.udiNumStations DO
				//Abort Station Sequence
				aStations[i].Stop();
			END_FOR
			sLog := CONCAT('Auto: End, State: ', INT_TO_STRING(iState));
			iState := 0;
		END_IF		
		
END_CASE
Automatic := bBusy;
END_METHOD

METHOD ConfigureStations : BOOL
VAR_INPUT
END_VAR
VAR_OUTPUT
END_VAR
VAR_INST
	bAllDone 	: BOOL;
	i			: UDINT;
END_VAR
bAllDone := TRUE;
FOR i:= 1 TO Tc3_XTS_Utility.TcIoXtsEnvironmentParameterList.MaxXtsInfoStation DO
	
	//Configure the relationship between stations
	IF i<stCfg.udiNumStations THEN
			aStations[i].configure(stCfg.stStationsCfg[i], udiNumMovers, lrPart1Length, ax[1].bMoverInverted, aStations[i+1]);
			//aStations[i].INextStation := aStations[i+1];	
	ELSIF i = stCfg.udiNumStations THEN	
			aStations[i].configure(stCfg.stStationsCfg[i], udiNumMovers, lrPart1Length, ax[1].bMoverInverted, aStations[1]);
			//aStations[i].INextStation := aStations[1];	
	ELSE
		aStations[i].configure(stCfg.stStationsCfg[i], udiNumMovers, lrPart1Length, ax[1].bMoverInverted, aStations[1]);
	END_IF

	//aStations[i](stCfg := stCfg.stStationsCfg[i], (*ax := ax,*) udiNumMovers := udiNumMovers, lrPartLength := lrPart1Length, bInvertPolarity := ax[1].bMoverInverted, ax := ax);
	IF stCfg.bNotCfgStationsViewer = FALSE THEN
		IF aStationsOTCID[i] <> 0 THEN
			bAllDone := bAllDone AND aStations[i].SetStationInfo(TRUE, OTCID := aStationsOTCID[i], i > SEL(stCurrentCfg.udiNumStations=0, stCurrentCfg.udiNumStations, stCfg.udiNumStations));
		END_IF
	ELSE
		bAllDone := TRUE;
	END_IF
END_FOR
IF bAllDone THEN
	FOR i:= 1 TO Tc3_XTS_Utility.TcIoXtsEnvironmentParameterList.MaxXtsInfoStation DO
		aStations[i].SetStationInfo(FALSE, OTCID := aStationsOTCID[i], FALSE);
	END_FOR
	ConfigureStations := TRUE;
END_IF
END_METHOD

METHOD cyclic : BOOL
VAR_INPUT
END_VAR
VAR
	i : UDINT;
END_VAR
//Initialization
Init(); 

//Operation
IF bInitDone THEN
	//Enable System
	bEnabled := Enable(bEnable);
	bInManual:= Manual(bManual AND bInAutomatic = FALSE AND bEnabled);
	bInAutomatic := Automatic(bAutomatic AND bInManual = FALSE AND bEnabled);
END_IF
Reset(bReset AND bAllMoversStandStill);

IF udiNumMovers <> 0 THEN
	//Call Group CA
	gp.Cyclic(ax);
	
	eGroupState 			:= gp.eGroupState;
	bAllMoversStandStill 	:= gp.bAllStandStill;
	
	//Call Movers
	FOR i := 1 TO TcIoXtsEnvironmentParameterList.MaxXtsMoversPerXpu DO
		ax[i].cyclic();
	END_FOR
	
	//Call Stations
	FOR i:= 1 TO stCfg.udiNumStations DO
		aStations[i].cyclic(ax);
	END_FOR
	
	//Status
	bReadyForMotion := gp.bGroupError = FALSE AND bEnabled;
	bError			:= gp.bGroupError;
END_IF
END_METHOD

METHOD PRIVATE Enable : BOOL
VAR_INPUT
	bEnable		: BOOL;
END_VAR
VAR_INST
	iState 		: INT;
	bAllDone 	: BOOL;
	i 			: UDINT;
	bDone		: BOOL;
END_VAR

IF (bError OR bReset) AND iState <> 999 AND iState <> 60 THEN iState := 999; END_IF

CASE iState OF
	
	0 : //Wait for Command
		IF bEnable THEN 
			FOR i := 1 TO udiNumMovers DO
				ax[i].ClearCmd();
			END_FOR
			gp.clearcmd();
			bDone := FALSE;
			iState := iState + 10; 
		END_IF
	
	10 : //Reset Movers
		sLog := CONCAT('Enable: Reset movers, State: ', INT_TO_STRING(iState));
		bAllDone := TRUE;
		FOR i := 1 TO udiNumMovers DO
			bAllDone := bAllDone AND ax[i].reset(TRUE).bDone;
		END_FOR
		IF bAllDone THEN
			iState := iState + 1;
		END_IF
		
	11 : //Power off all
		sLog := CONCAT('Disable: Power off all movers, State: ', INT_TO_STRING(iState));
		bAllDone := TRUE;
		FOR i := 1 TO udiNumMovers DO
			bAllDone := bAllDone AND ax[i].power_off().bDone;
		END_FOR
		IF bAllDone THEN
			iState := iState + 1;
		END_IF
		
	12 : //Configure movers inversion
		sLog := CONCAT('Enable: Configure movers inversion, State: ', INT_TO_STRING(iState));
		bAllDone := TRUE;
		FOR i := 1 TO udiNumMovers DO
			bAllDone := bAllDone AND ax[i].InvertPolarity(TRUE, stCfg.bInvertPolarity);
		END_FOR
	 	IF bAllDOne THEN
			 FOR i := 1 TO udiNumMovers DO
			 	ax[i].InvertPolarity(FALSE, stCfg.bInvertPolarity);
		 	 END_FOR
			 iState := 20;
	 	END_IF
		
	20 : //Power all Axis
		sLog := CONCAT('Enable: Power on movers, State: ', INT_TO_STRING(iState));
		bAllDone := TRUE;
		FOR i := 1 TO udiNumMovers DO
			bAllDone := bAllDone AND ax[i].power_on().bDone;
			IF ax[i].power_on().bError THEN
				sLog := CONCAT('Enable: Power on movers errors on mover: ', UDINT_TO_STRING(i));
				sLog := CONCAT(sLog, UDINT_TO_STRING(ax[i].power_on().udiErrorID));
				EXIT;
				iState := 999;
			END_IF
		END_FOR
		IF bAllDone THEN
			iState := iState + 1;
		END_IF
		
	21 : //Decopule axis
		sLog := CONCAT('Enable: Gear out movers, State: ', INT_TO_STRING(iState));
		FOR i:=1 TO udiNumMovers DO
			IF ax[i].p_Axis.Status.Coupled  THEN
				//
				bAllDone := bAllDOne AND ax[i].gearOut(TRUE).bDone;
			END_IF
		END_FOR
		IF bAllDOne THEN
			FOR i:=1 TO udiNumMovers DO
				ax[i].gearOut(FALSE);
			END_FOR
			iState := 30;
		END_IF
		
	30 : //Reset Group
		sLog := CONCAT('Enable: Reset group CA, State: ', INT_TO_STRING(iState));
		IF gp.reset(TRUE).bDone THEN
			iState := iState + 10;
		ELSIF gp.reset(TRUE).bError THEN
			sLog := CONCAT('Enable: Reset group CA Error : ', UDINT_TO_STRING(gp.reset(TRUE).udiErrorID));
			gp.reset(FALSE);
			iState := 1000;
		END_IF
		
	40 : //Add all axis to group
		sLog := CONCAT('Enable: Add movers to group, State: ', INT_TO_STRING(iState));
		bAllDone := TRUE;
		FOR i := 1 TO udiNumMovers DO
			bAllDone := bAllDone AND ax[i].add2Group(TRUE, ag := gp.ag).bDone;
		END_FOR
		IF bAllDone THEN
			FOR i := 1 TO udiNumMovers DO
				ax[i].add2Group(FALSE, ag := gp.ag);
			END_FOR
			iState := iState + 10;
		END_IF
		
	50 : //Enable group
		sLog := CONCAT('Enable: Enable group CA, State: ', INT_TO_STRING(iState));
		IF gp.enable(TRUE).bDone THEN
			iState := iState + 10;
			sLog := CONCAT('Enable: Enable done!, State: ', INT_TO_STRING(iState));
		ELSIF gp.enable(TRUE).bError THEN
			sLog := CONCAT('Enable: Enable group CA Error : ', UDINT_TO_STRING(gp.enable(TRUE).udiErrorID));
			gp.enable(FALSE);
			iState := 1000;
		END_IF
		
	60 : //Jog Done
		 bDone := TRUE;
		 IF bEnable = FALSE THEN iState := 70; END_IF 

	70 : //Halt group
		sLog := CONCAT('Disable: Halt movers, State: ', INT_TO_STRING(iState));
		bAllDone := TRUE;
		FOR i := 1 TO udiNumMovers DO
			bAllDone := bAllDone AND ax[i].haltca(TRUE).bDone;
		END_FOR
		IF bAllDone THEN
			iState := iState + 10;
		END_IF
		
	80 : //Disable
		sLog := CONCAT('Disable: Disable group CA, State: ', INT_TO_STRING(iState));
		IF gp.disable(TRUE).bDone THEN
			iState := iState + 10;
		ELSIF gp.disable(TRUE).bError THEN
			sLog := CONCAT('Disable: Disable group CA Error : ', UDINT_TO_STRING(gp.disable(TRUE).udiErrorID));
			gp.disable(FALSE);
			iState := 1000;
		END_IF		

	90 : //UnGroup
		sLog := CONCAT('Disable: Ungroup all movers, State: ', INT_TO_STRING(iState));
		IF gp.ungroupall(TRUE).bDone THEN
			iState := iState + 10;
		ELSIF gp.ungroupall(TRUE).bError THEN
			sLog := CONCAT('Disable: UnGroup all movers Error : ', UDINT_TO_STRING(gp.ungroupall(TRUE).udiErrorID));
			gp.ungroupall(FALSE);
			iState := 1000;
		END_IF
	
	100 : //Power off all
		sLog := CONCAT('Disable: Power off all movers, State: ', INT_TO_STRING(iState));
		bAllDone := TRUE;
		FOR i := 1 TO udiNumMovers DO
			bAllDone := bAllDone AND ax[i].power_off().bDone;
		END_FOR
		IF bAllDone THEN
			sLog := 'Disable: Done!';
			bDone := FALSE;
			iState := 0;
		END_IF
		
	999 : //Abort
		sLog := CONCAT('Enable: Abort, State: ', INT_TO_STRING(iState));
		iState := 0;
		
	1000 : //Error
		iState := 0;
		 
END_CASE
Enable := bDone;
END_METHOD

METHOD PRIVATE Init
VAR_INST
	iState 		: INT;
	bAllDone 	: BOOL;
	i 			: UDINT;
	udiErrorID	: UDINT;
	bSomeError  : BOOL;
END_VAR

//XPU Initialization
IF bXPUInitDone = FALSE THEN
	sLog := 'Init: Initialazing XPU';
	IF fbXTSEnv.Init(TRUE) THEN
		sLog := 'Init: XPU Initialazed';
		fbXTSEnv.Init(FALSE);
		bXPUInitDone := TRUE;
	END_IF	
END_IF

IF bReset AND iState <> 999 AND bInitDone = FALSE THEN iState := 999; END_IF

CASE iState OF
	
	0 : 
		IF bXPUInitDone THEN 
			gp.clearCmd();
			FOR i:=1 TO udiNumMovers DO
				bAllDone := bAllDOne AND ax[i].clearCmd();
			END_FOR
			iState := iState + 10; 
		END_IF
	
	10 : //Get XPU Parameters
		sLog := 'Init: Checking XPU parameters';
		Ixpu 						:= fbXTSEnv.XpuTcIo(1);
		IPart1						:= Ixpu.PartTcIo(1);
		iOperationMode 				:= Ixpu.GetOperationMode();
		AreAllPositionValid 		:= Ixpu.GetAreAllPositionsValid();
		DetectedMoverCount 			:= Ixpu.GetDetectedMoverCount();
		ExpectedMoverCount 			:= Ixpu.GetExpectedMoverCount();
		HasMoverIDDetectorError 	:= Ixpu.GetHasMoverIdDetectionError();
		IsMoveriddetectoractive 	:= Ixpu.GetIsMoverIdDetectionActive();
		ismoverisdetectionvalid 	:= Ixpu.GetIsMoverIdDetectionValid();
		TrackCount					:= Ixpu.GetTrackCount();
		PartCount					:= Ixpu.GetPartCount();
		lrPart1Length 				:= IPart1.GetLength();
		udiPart1NumModules			:= IPart1.GetModuleCount();
		udiNumMovers 				:= Ixpu.GetMoverCount();
		eMoverType					:= Ixpu.GetMoverType();
		
		IF (Ixpu.GetDetectedMoverCount() = Ixpu.GetExpectedMoverCount()) AND Ixpu.GetAreAllPositionsValid() THEN
			iState := iState + 10; 			
		END_IF

	20 : //Detect Mover 1 
		sLog := 'Init: Detecting mover 1';
		IF Ixpu.GetIsMoverIdDetectionValid() = FALSE THEN
			IF Ixpu.GetMoverIdDetectionMode() = 1 THEN
				Ixpu.TriggerMoverIdDetection();
				iState := iState + 1;
			ELSE
				bMover1DetectionValid := TRUE;
				iState := iState + 10;
			END_IF
		ELSE
			bMover1DetectionValid := TRUE;
			iState := iState + 10;
		END_IF
		
	21 : //Check Mover 1 Detection Valid
		IF Ixpu.GetIsMoverIdDetectionValid() THEN
			bMover1DetectionValid := TRUE;
			iState := 30;
		END_IF
	
	30 : //Get OIDS of Group CA
		sLog := 'Init: Getting group CA Oids';
		IF fbXTSEnv.GetCaGroupOids(TRUE) THEN
			fbXTSEnv.GetCaGroupOids(FALSE);
			GroupCAOTCID := fbXTSEnv.P_CaGroupOids;
			IF gp.init(TRUE, GroupCAOTCID[1]) THEN
				gp.init(FALSE, GroupCAOTCID[1]);
				iState := 31;
			END_IF
		END_IF
		
	31 : //Reset Group
		sLog := 'Init: Reset group CA';
		IF gp.reset(TRUE).bDone THEN
			gp.reset(FALSE);
			iState := iState + 1;
		ELSIF gp.reset(TRUE).bError THEN
			sLog := CONCAT('Init: Reset group CA Error : ', UDINT_TO_STRING(gp.reset(TRUE).udiErrorID));
			gp.reset(FALSE);
			iState := 1000;
		END_IF
		
	32 : //Disable Group in order to configure the Rail Length
		sLog := 'Init: UnGroup all';
		IF gp.ungroupall(TRUE).bDone THEN
			gp.ungroupall(FALSE);
			iState := iState + 1;
		ELSIF gp.ungroupall(TRUE).bError THEN
			sLog := CONCAT('Init: UnGroup all movers Error : ', UDINT_TO_STRING(gp.ungroupall(TRUE).udiErrorID));
			gp.ungroupall(FALSE);
			iState := 1000;
		END_IF
		
	33 : //Set Group CA Rail Length equal to Part 1 length
		sLog := 'Init: Get group CA Oids';
		//IF gp.fbXPUGroupCA.Init(TRUE, GroupCAOTCID[1]) THEN
			IF gp.SetRailLength(lrPart1Length) THEN
				//gp.fbXPUGroupCA.Init(FALSE, GroupCAOTCID[1]);
				iState := 40;		
			END_IF
		//END_IF
		
	40 : //Get Info Server OIDS
		sLog := 'Init: Get Info Server Oids';
		IF Tc3_XTS_Utility.TcIoXtsEnvironmentParameterList.MaxXtsInfoServer > 0 THEN 
			IF fbXTSEnv.GetInfoServerOids(TRUE) THEN
				fbXTSEnv.GetInfoServerOids(FALSE);
				aInfoServerOids := fbXTSEnv.P_InfoServerOids;
				i:=1;
				fbInfoServer.Init(FALSE, aInfoServerOids[i]);
				iState := iState + 1;
			END_IF
		ELSE
			iState := iState + 10;
		END_IF

	41 : //Get OCID of Stations
		sLog := 'Init: Get Info Stations Oids';
		IF fbInfoServer.Init(TRUE, aInfoServerOids[i]) THEN
			IF fbInfoServer.GetInfoStationOids() THEN
				aStationsOTCID := fbInfoServer.P_InfoStationOids;
				fbInfoServer.Init(FALSE, aInfoServerOids[i]);
				FOR i:= 1 TO stCfg.udiNumStations DO
					aStations[i].SetStationInfo(FALSE, OTCID := aStationsOTCID[i], FALSE);
				END_FOR
				iState := 50;
			END_IF
		END_IF
		
	50 : //Get Mover OIDS
		sLog := 'Init: Get movers Oids';
		IF IXPU.GetMoverOids() THEN
			aMoversOids := IXPU.P_MoverOids;
			iState := iState + 1;
		END_IF
		
	51 : //Gear out movers
		sLog := 'Init: Gear out movers';
		bAllDone := TRUE;
		FOR i:=1 TO udiNumMovers DO
			IF ax[i].p_Axis.Status.Coupled THEN
				//
				bAllDone := bAllDOne AND ax[i].gearOut(TRUE).bDone;
			END_IF
		END_FOR
		IF bAllDOne THEN
			FOR i:=1 TO udiNumMovers DO
				ax[i].gearOut(FALSE);
			END_FOR
			iState := iState + 1;
		END_IF
		
	52 : //Reset Movers
		sLog := 'Init: Reset movers';
		bAllDOne := TRUE;
		 FOR i := 1 TO udiNumMovers DO
			bAllDone := bAllDone AND ax[i].reset(TRUE).bDone;
			IF ax[i].reset(TRUE).bError THEN
				bSomeError := TRUE; 
				EXIT; 
			END_IF
		 END_FOR
		 IF bAllDOne THEN
			 FOR i := 1 TO udiNumMovers DO
			 	ax[i].reset(FALSE);
		 	 END_FOR
			 iState := iState + 1;
		 ELSIF bSomeError THEN
			sLog := CONCAT('Init: Reset movers Error in mover : ', UDINT_TO_STRING(i));
			sLog := CONCAT('sLog: ', UDINT_TO_STRING(ax[i].reset(TRUE).udiErrorID));
			FOR i := 1 TO udiNumMovers DO
			 	ax[i].reset(FALSE);
		 	 END_FOR
			bSomeError 	:= FALSE;
			iState 		:= 1000;
		 END_IF
		 
	53 : //Power off Movers
		sLog := 'Init: Power off movers';
		bAllDOne := TRUE;
		 FOR i := 1 TO udiNumMovers DO
			 bAllDone := bAllDone AND ax[i].power_off().bDone;
		 END_FOR
		 IF bAllDOne THEN
			 iState := iState + 1;
		 END_IF
		 
	54 : //Configure Movers
		sLog := 'Init: Configure movers';
		 bAllDone := TRUE;
		 FOR i := 1 TO udiNumMovers DO
			 bAllDone := bAllDone AND ax[i].InvertPolarity(TRUE, stCfg.bInvertPolarity);
		 END_FOR
	 	IF bAllDOne THEN
			 FOR i := 1 TO udiNumMovers DO
			 	ax[i].InvertPolarity(FALSE, stCfg.bInvertPolarity);
		 	 END_FOR
			 iState := 55;
	 	END_IF
		
	55 : //Init Movers
		bAllDone := TRUE;
		 FOR i := 1 TO udiNumMovers DO
			 bAllDone := bAllDone AND ax[i].Init(TRUE, aMoversOids[i]);
		 END_FOR
		 IF bAllDOne THEN
			 FOR i := 1 TO udiNumMovers DO
			 	ax[i].Init(FALSE, aMoversOids[i]);
		 	 END_FOR
		 	iState := 60;
		 END_IF
		
	60 : //Init Stations
		bAllDone := TRUE;
		FOR i:= 1 TO stCfg.udiNumStations DO
			aStations[i].Init(TRUE, aStationsOTCID[i]);
		END_FOR
		IF bAllDone THEN
			FOR i:= 1 TO stCfg.udiNumStations DO
				aStations[i].Init(FALSE, aStationsOTCID[i]);
			END_FOR
			iState := iState + 1;
		END_IF
		
	61 : //Set Stations configuration
		sLog := 'Init: Configure stations';
		IF ConfigureStations() THEN
			stVisuStationsCfg := stCfg.stStationsCfg;
			iState := 70;
		END_IF
		
	70 : //Jog Done
		 sLog := 'Init: Done!';
		 bInitDone 	:= TRUE;
		 iState := 71;
		 
	71 :
		//
		
	999: //Abort
		sLog := CONCAT('Init: Abort, State: ', INT_TO_STRING(iState));
		iState := 0;
		
	1000 : //Error
		iState := 0;
			 
END_CASE
END_METHOD

METHOD IsPassiveMover : BOOL
VAR_INPUT
	ID 				: UDINT;
END_VAR
VAR_INST
	i 				: DINT;
	bFirstMoverEven : BOOL;
	iTmp			: udint;
END_VAR
IF stCFg.udiMoverMode = 2 THEN
	bFirstMoverEven := (udiFirstMover MOD 2) = 0;
	IsPassiveMover := ((ID MOD 2) <> 0 AND bFirstMoverEven) OR ((ID MOD 2) = 0 AND bFirstMoverEven = FALSE);
ELSIF stCFg.udiMoverMode = 3 THEN
	iTmp := udiFirstMover MOD 3;
	IsPassiveMover := ((ID MOD 3) <> iTmp); //AND bFirstMoverEven) OR ((ID MOD 3) <> 0 AND bFirstMoverEven = FALSE);
END_IF

	(*i := udiFirstMover-1;
	WHILE i = udiFirstMover+1 DO
		//
		IF ID = DINT_TO_UDINT(i) THEN 
			m_isPassiveMover := TRUE; 
			RETURN;
		END_IF
		i := i - 2;
		IF i < 1 THEN i := stCfg.uiTotalAxis; END_IF
	END_WHILE*)

	(*FOR i := udiFirstMover-1 TO 1 BY -2 DO
		IF ID = DINT_TO_UDINT(i) THEN 
			m_isPassiveMover := TRUE; 
			RETURN;
		END_IF	
		IF i < 1 THEN
			RETURN;
		END_IF
	END_FOR	
	
	FOR i := stCfg.uiTotalAxis TO udiFirstMover BY -2 DO
		IF ID = DINT_TO_UDINT(i) THEN 
			m_isPassiveMover := TRUE; 
			RETURN;
		END_IF	
		IF i < 1 THEN
			RETURN;
		END_IF
	END_FOR*)

//END_IF
END_METHOD

METHOD PRIVATE Manual : BOOL
VAR_INPUT
	bEnable 			: BOOL;
END_VAR
VAR_INST
	iState 				: INT;
	bAllDone 			: BOOL;
	i 					: UDINT;
	bBusy				: BOOL;
	fbRTRIG				: R_Trig;
	m_udiStationSelection : UDINT;
END_VAR

IF (bError OR bReset) AND iState <> 999 and bBusy THEN iState := 999; END_IF

CASE iState OF
	0 : IF bEnable THEN 
			iState := iState + 1; 
			bBusy  := TRUE;
		END_IF
		
	1 : //Idle
		sLog := CONCAT('Manual: Idle, State: ', INT_TO_STRING(iState));
		
		IF iVisuMoverSelection > 0 THEN udiMoverSelection := INT_TO_UDINT(iVisuMoverSelection); ELSE udiMoverSelection := 0; END_IF
		IF iVisuStationSelection > 0 THEN udiStationSelection := INT_TO_UDINT(iVisuStationSelection); ELSE udiStationSelection := 0; END_IF
		IF iVisuStopPositionSelection > 0 THEN udiStopPositionSelection	:= INT_TO_UDINT(iVisuStopPositionSelection); ELSE udiStopPositionSelection := 0; END_IF
		
		IF bEnable = FALSE THEN
			iState := 100;
		ELSIF bJogBackwards OR bJogForward THEN
			iState := 10; 
		ELSIF bManualMove AND udiStationSelection = 0 THEN
			//Move All with Target Position
			iState := 50; 
		ELSIF bManualMove AND udiStationSelection > 0 AND udiStationSelection < stCfg.udiNumStations+1 AND udiStopPositionSelection > 0 AND udiStopPositionSelection < 6 THEN
			//Move Mover to Station 
			iState := 60;
		ELSIF bTeachStation AND udiStationSelection > 0 AND udiMoverSelection > 0 AND udiStopPositionSelection > 0 AND udiStopPositionSelection < 6 THEN
			m_udiStationSelection := udiStationSelection;
			iState := 70;
		END_IF
		
	10 : //Manual mode operation 0 
		sLog := CONCAT('Manual: Jogging, State: ', INT_TO_STRING(iState));
		IF udiMoverSelection = 0 THEN
			bAllDone := TRUE;
			FOR i := 1 TO udiNumMovers DO
				bAllDone := bAllDone AND ax[i].jogca_velo(bJogBackwards, bJogForward, lrTargetVelocity).bBusy = FALSE;
			END_FOR
			IF bJogBackwards = FALSE AND bJogForward = FALSE AND bAllDone THEN
				iState := 1;
			END_IF	
		ELSE
			IF udiMoverSelection < 1 OR udiMoverSelection > udiNumMovers THEN udiMoverSelection := 1; END_IF
			IF ax[udiMoverSelection].jogca_velo(bJogBackwards, bJogForward, lrTargetVelocity).bBusy = FALSE AND bJogBackwards = FALSE AND bJogForward = FALSE THEN
				iState := 1;	
			END_IF
		END_IF
		
	50 : //Manual Operation with Target Position
		sLog := CONCAT('Manual: Go to target position: ', INT_TO_STRING(iState));
		IF udiMoverSelection = 0 THEN
			FOR i := 1 TO udiNumMovers DO
				ax[i].moveca_direction(bManualMove, lrTargetPosition, lrTargetVelocity, Direction);
			END_FOR
			IF bAllMoversStandStill AND bManualMove = FALSE THEN
				iState := 1;
			END_IF
		ELSE ax[udiMoverSelection].moveca_direction(bManualMove, lrTargetPosition, lrTargetVelocity, Direction);
			IF bAllMoversStandStill AND bManualMove = FALSE THEN
				iState := 1;
			END_IF
		END_IF
		
	60 : //Manual Operation with Stations
		sLog := CONCAT('Manual: Go to station: ', INT_TO_STRING(iState));
		IF udiMoverSelection = 0 THEN
			FOR i := 1 TO udiNumMovers DO
				IF udiStopPositionSelection = 1 THEN
					ax[i].moveca_direction(bManualMove, aStations[udiStationSelection].stCfg.lrStartPosition, lrTargetVelocity, Direction);		
				ELSIF udiStopPositionSelection > 1 AND udiStopPositionSelection < 5 THEN
					ax[i].moveca_direction(bManualMove, aStations[udiStationSelection].stCfg.lrStopPosition[udiStopPositionSelection-1] + aStations[udiStationSelection].stCfg.lrStartPosition, lrTargetVelocity, Direction);					
				ELSIF udiStopPositionSelection = 5 THEN
					ax[i].moveca_direction(bManualMove, aStations[udiStationSelection].stCfg.lrEndPosition, lrTargetVelocity, Direction);	
				END_IF
			END_FOR
			IF bAllMoversStandStill AND bManualMove = FALSE THEN
				iState := 1;
			END_IF
		ELSE 
			IF udiStopPositionSelection = 1 THEN
				ax[udiMoverSelection].moveca_direction(bManualMove, aStations[udiStationSelection].stCfg.lrStartPosition, lrTargetVelocity, Direction);		
			ELSIF udiStopPositionSelection > 1 AND udiStopPositionSelection < 5 THEN
				ax[udiMoverSelection].moveca_direction(bManualMove, aStations[udiStationSelection].stCfg.lrStopPosition[udiStopPositionSelection-1] + aStations[udiStationSelection].stCfg.lrStartPosition, lrTargetVelocity, Direction);					
			ELSIF udiStopPositionSelection = 5 THEN
				ax[udiMoverSelection].moveca_direction(bManualMove, aStations[udiStationSelection].stCfg.lrEndPosition, lrTargetVelocity, Direction);	
			END_IF
			IF bAllMoversStandStill AND bManualMove = FALSE THEN
				iState := 1;
			END_IF
		END_IF
		
	70 : //Teach Station
		sLog := CONCAT('Manual: Teaching station: ', INT_TO_STRING(iState));
		IF udiStopPositionSelection = 1 THEN
			stCfg.stStationsCfg[m_udiStationSelection].lrStartPosition := ax[udiMoverSelection].p_Axis.NcToPlc.ModuloSetPos;		
		ELSIF udiStopPositionSelection > 1 AND udiStopPositionSelection < 5 THEN
			stCfg.stStationsCfg[m_udiStationSelection].lrStopPosition[udiStopPositionSelection-1] := ax[udiMoverSelection].p_Axis.NcToPlc.ModuloSetPos-stCfg.stStationsCfg[m_udiStationSelection].lrStartPosition;					
		ELSIF udiStopPositionSelection = 5 THEN
			stCfg.stStationsCfg[m_udiStationSelection].lrEndPosition := ax[udiMoverSelection].p_Axis.NcToPlc.ModuloSetPos;			
		END_IF
		IF ConfigureStations() THEN iState := iState + 1; END_IF
		
	71 : //Apply New Configuration
		sLog := CONCAT('Manual: Teaching done: ', INT_TO_STRING(iState));
		bTeachDone := TRUE;
		IF bTeachStation = FALSE THEN
			bTeachDone := FALSE;
			iState := 1;
		END_IF
		
	100 : 
		sLog := CONCAT('Manual: End, State: ', INT_TO_STRING(iState));
		bBusy := FALSE;
		iState := 0;
		
	999 : //Abort
		sLog := CONCAT('Manual: Abort, State: ', INT_TO_STRING(iState));
		bBusy := FALSE;
		iState := 0;
		
END_CASE
Manual := bBusy;
END_METHOD

METHOD Reset : BOOL
VAR_INPUT
	bEnable 	: BOOL;
END_VAR
VAR_INST
	iState		: INT;
	i 			: UDINT;
	bAllDOne 	: BOOL;
END_VAR

IF bEnable = FALSE THEN iState := 0; END_IF

CASE iState OF
	0 : IF bEnable THEN 
			FOR i:=1 TO udiNumMovers DO
				ax[i].reset(FALSE);
				ax[i].gearOut(FALSE);
			END_FOR
			gp.reset(FALSE);
			iState := iState + 1; 
		END_IF
	1 :
		bAllDone := TRUE;
		FOR i:=1 TO udiNumMovers DO
			IF ax[i].p_Axis.Status.Coupled = FALSE THEN
				bAllDone := bAllDOne AND ax[i].reset(TRUE).bDone;
			END_IF
		END_FOR
		IF bAllDone THEN
			FOR i:=1 TO udiNumMovers DO
				bAllDone := bAllDOne AND ax[i].reset(FALSE).bDone;
			END_FOR
			iState := iState + 1;
		END_IF
		
	2 : //Check if there is some axis coupled and decoupled (Is not possible to perform a reset group with axis coupled)
		bAllDone := TRUE;
		FOR i:=1 TO udiNumMovers DO
			IF ax[i].p_Axis.Status.Coupled THEN
				//
				bAllDone := bAllDOne AND ax[i].gearOut(TRUE).bDone;
			END_IF
		END_FOR
		IF bAllDOne THEN
			FOR i:=1 TO udiNumMovers DO
				ax[i].gearOut(FALSE);
			END_FOR
			iState := iState + 1;
		END_IF
	
	3 : //Reset Group
		IF gp.reset(TRUE).bDone THEN
			iState := iState + 1;
			gp.reset(FALSE);
		ELSIF gp.reset(TRUE).bError THEN
			sLog := CONCAT('Reset: Reset group CA Error : ', UDINT_TO_STRING(gp.reset(TRUE).udiErrorID));
			gp.reset(FALSE);
			iState := 1000;
		END_IF
		
	4 : //Reset Done
		Reset := TRUE;
		IF bEnable = FALSE THEN
			iState := 0;
		END_IF
		
	1000 : //Error
		iState := 0;
END_CASE
END_METHOD

METHOD WhoIsAtPos : UDINT
VAR_INPUT
	lrPosition : LREAL;
END_VAR
VAR_INST
	i 			: UDINT;
	lrDistance	: LREAL;
END_VAR
FOR i := 1 TO udiNumMovers DO
	lrDistance := lrPosition - ax[i].p_ModulePos;
	IF ABS(lrDistance) < 1.0 OR ABS(lrDistance - lrPart1Length) < 1.0 THEN
		WhoIsAtPos := ax[i].udiID;
	END_IF
END_FOR
END_METHOD

END_FUNCTION_BLOCK

// ---- POUs/XTS/Movers/FB_Mover.TcPOU
FUNCTION_BLOCK FB_Mover EXTENDS FB_TcIoXtsXPUMover
VAR_OUTPUT
	udiID					: UDINT;
	bMoverInverted			: BOOL;
END_VAR
VAR
	ax						: AXIS_REF;
	fbPower 				: MC_Power;
	fbReset 				: MC_Reset;
	fbHaltCA				: MC_HaltCA;
	fbMoveAbsCA				: MC_MoveAbsoluteCA;
	fbMoveRelCA				: MC_MoveRelativeCA;
	fbMoveAbsTimeCA			: MC_MoveAbsoluteTimeCA;
	fbMoveAbs				: MC_MoveAbsolute;
	fbGearIn				: MC_GearIn;
	fbGearOut				: MC_GearOut;
	fbReadParamSet			: MC_ReadParameterSet := (Execute := TRUE);
	fbAddAxis2Group 		: MC_AddAxisToGroup;
	stParameter				: ST_AxisParameterSet;
	fbJogCA					: MC_JOGCA;
	fbJog					: MC_Jog;
	bInternalControl		: BOOL;
	lrTargetPos				: LREAL;
	bTmp					: BOOL;
END_VAR

METHOD add2Group : REFERENCE TO stFeedback
VAR_INPUT
	bExecute	: BOOL;
	ag		 	: AXES_GROUP_REF;
END_VAR
VAR_INST
	stStatus	: stFeedback;
END_VAR
fbAddAxis2Group(
	AxesGroup:= ag, 
	Axis:= ax, 
	Execute:= bExecute, 
	IdentInGroup:= UDINT_TO_IDENTINGROUP(ax.NcToPlc.AxisId), 
	Done=> stStatus.bDone, 
	Busy=> stStatus.bBusy, 
	Error=> stStatus.bError, 
	ErrorId=> stStatus.udiErrorID);
	
add2Group REF= stStatus;
END_METHOD

METHOD clearCmd : BOOL
VAR_INPUT
END_VAR
fbMoveAbsCA.Execute := FALSE;
fbHaltCA.Execute := FALSE;
fbGearIn.Execute := FALSE;
fbReset.Execute	:= FALSE;
fbMoveAbsTimeCA(Axis := ax, bExecute := FALSE);
fbGearIn(master := ax, slave := ax, Execute := FALSE);
fbGearOut(slave := ax, Execute := FALSE);
InvertPolarity(FALSE, FALSE);
END_METHOD

METHOD cyclic : BOOL
VAR_INPUT
END_VAR
ax.ReadStatus();

fbPower(
	Axis:= ax, 
	Enable:= , 
	Enable_Positive:= , 
	Enable_Negative:= , 
	Override:= , 
	BufferMode:= , 
	Options:= , 
	Status=> , 
	Busy=> , 
	Active=> , 
	Error=> , 
	ErrorID=> );
	
fbReset(
	Axis:= ax, 
	Execute:= , 
	Busy=> , 
	Done=> ,
	Error=> , 
	ErrorID=> );
	
fbJog(
	Axis:= ax, 
	JogForward:= , 
	JogBackwards:= , 
	Mode:= , 
	Position:= , 
	Velocity:= , 
	Acceleration:= , 
	Deceleration:= , 
	Jerk:= , 
	Done=> , 
	Busy=> , 
	Active=> , 
	CommandAborted=> , 
	Error=> , 
	ErrorID=> );

fbJogCA(
	Axis:= ax, 
	JogForward:= , 
	JogBackwards:= , 
	Mode:= , 
	Position:= , 
	Velocity:= , 
	Acceleration:= , 
	Deceleration:= , 
	Jerk:= , 
	Done=> , 
	Busy=> , 
	Active=> , 
	CommandAborted=> , 
	Error=> , 
	ErrorID=> );
	
fbMoveAbsCA(
	Axis:= ax, 
	Execute:= , 
	ContinuousUpdate:= , 
	Position:= , 
	Velocity:= , 
	Acceleration:= , 
	Deceleration:= , 
	Jerk:= , 
	Gap:= , 
	BufferMode:= , 
	Direction:= , 
	Options:= , 
	Busy=> , 
	Done=> ,
	Error=> , 
	ErrorID=> );
	
fbMoveAbsTimeCA(
	Axis:= ax, 
	bExecute:= , 
	lrPosition:= , 
	lrTime:= , 
	Done=> , 
	Busy=> , 
	Active=> , 
	CommandAborted=> , 
	Error=> , 
	ErrorId=> );
	
fbHaltCA(
	Axis:= ax, 
	Execute:= , 
	Deceleration:= , 
	Jerk:= , 
	Options:= , 
	Busy=> , 
	Done=> ,
	Error=> , 
	ErrorID=> );

fbMoveAbs(
	Axis:= ax, 
	Execute:= , 
	Position:= , 
	Velocity:= , 
	Acceleration:= , 
	Deceleration:= , 
	Jerk:= , 
	BufferMode:= , 
	Options:= , 
	Busy=> , 
	Done=> ,
	Error=> , 
	ErrorID=> );
	
fbMoveRelCA(
	Axis:= ax, 
	Execute:= , 
	ContinuousUpdate:= , 
	Distance:= , 
	Velocity:= , 
	Acceleration:= , 
	Deceleration:= , 
	Jerk:= , 
	Gap:= , 
	BufferMode:= , 
	Options:= , 
	Busy=> , 
	Done=> ,
	Error=> , 
	ErrorID=> );
	
fbGearOut(
	Slave:= ax, 
	Execute:= , 
	Options:= , 
	Done=> , 
	Busy=> , 
	Error=> , 
	ErrorID=> );

fbReadParamSet(Parameter := stParameter, Axis := ax);
udiID := stParameter.AxisId;
END_METHOD

METHOD gearIn : REFERENCE TO stFeedback
VAR_INPUT
	bExecute 			: BOOL;
	lrRatioNumerator 	: LREAL;
	uiRatioDenominator	: UINT;
END_VAR
VAR_IN_OUT
	axMaster	: AXIS_REF;	
END_VAR
VAR_INST
	stStatus	: stFeedback;
END_VAR
fbGearIn.Execute 	:= bExecute;

fbGearIn(
	Master:= axMaster, 
	Slave:= ax, 
	Execute:= , 
	RatioNumerator:= lrRatioNumerator, 
	RatioDenominator:= uiRatioDenominator, 
	Acceleration:= , 
	Deceleration:= , 
	Jerk:= , 
	BufferMode:= , 
	Options:= , 
	InGear=> stStatus.bDone, 
	Busy=> stStatus.bBusy, 
	Active=> , 
	CommandAborted=> stStatus.bCommandAborted, 
	Error=> stStatus.bError, 
	ErrorID=> stStatus.udiErrorID);
	
gearin REF= stStatus;
END_METHOD

METHOD gearOut : REFERENCE TO stFeedback
VAR_INPUT
	bExecute 			: BOOL;
END_VAR
VAR_INST
	stStatus : stFeedback;
END_VAR
fbGearOut.Execute 	:= bExecute;
stStatus.bDone		:= fbGearOut.Done;
stStatus.bBusy		:= fbGearOut.Busy;
stStatus.bError		:= fbGearOut.Error;
stStatus.udiErrorID	:= fbGearOut.ErrorID;

gearout REF= stStatus;
END_METHOD

METHOD getmoveratpos : BOOL
VAR_INPUT
	lrPosition : LREAL;
END_VAR
IF ax.NcToPlc.ModuloSetPos > lrPosition-1 AND ax.NcToPlc.ModuloSetPos < lrPosition+1 THEN
	getmoveratpos := TRUE;
END_IF
END_METHOD

METHOD haltca : REFERENCE TO stFeedback
VAR_INPUT
	bExecute : BOOL;
END_VAR
VAR_INST
	stStatus : stFeedback;
END_VAR
fbHaltCA.Execute 	:= bExecute;
fbHaltCA.Gap		:= MC_DEFAULT;
stStatus.bDone		:= fbHaltCA.Done;
stStatus.bBusy		:= fbHaltCA.Busy;
stStatus.bError		:= fbHaltCA.Error;
stStatus.udiErrorID	:= fbHaltCA.ErrorID;

haltca REF= stStatus;
END_METHOD

METHOD InvertPolarity : BOOL
VAR_INPUT
	bExecute : BOOL;
	bValue	 : BOOL;
END_VAR
VAR_INST
	iState 		: INT;
	fbWrite 	: MC_WriteParameterPersistent;
END_VAR

CASE iState OF 
	0 : IF bExecute THEN 
			fbWrite(Axis := ax, Execute := FALSE);
			iState := iState + 1; 
		END_IF
	1 :  
		fbWrite(
			Axis:= ax, 
			Execute:= TRUE, 
			ParameterNumber:= MC_AxisParameter.AxisMotorDirectionInverse, 
			Value:= BOOL_TO_LREAL(bValue), 
			Done=> , 
			Busy=> , 
			Error=> , 
			ErrorID=> );
		IF fbWrite.Done THEN
			fbWrite(Axis := ax, Execute := FALSE);
			iState := iState + 1;
		END_IF
		IF fbWrite.Error THEN
			iState := 999;
		END_IF
		
	2 : 
		fbWrite(
			Axis:= ax, 
			Execute:= TRUE, 
			ParameterNumber:= MC_AxisParameter.AxisEncoderDirectionInverse, 
			Value:= BOOL_TO_LREAL(bValue), 
			Done=> , 
			Busy=> , 
			Error=> , 
			ErrorID=> );
		IF fbWrite.Done THEN
			fbWrite(Axis := ax, Execute := FALSE);
			iState := iState + 1;
		END_IF
		IF fbWrite.Error THEN
			iState := 999;
		END_IF
		
	3 : //Job Done
		InvertPolarity := TRUE;
		bMoverInverted := bValue;
		IF bExecute = FALSE THEN
			iState := 0;
		END_IF
		
	999 : //Error
		iState := 0;
		
END_CASE
END_METHOD

METHOD jogca : REFERENCE TO stFeedback
VAR_INPUT
	bJogBackwards	: BOOL;
	bJogForward		: BOOL;
END_VAR
VAR_INST
	stStatus		: stFeedback;
END_VAR
fbJogCA.JogBackwards			:= bJogBackwards;
fbJogCA.JogForward				:= bJogForward;

stStatus.bDone					:= fbJogCA.Done;
stStatus.bBusy					:= fbJogCA.Busy;
stStatus.bCommandAborted		:= fbJogCA.CommandAborted;
stStatus.bError					:= fbJogCA.Error;
stStatus.udiErrorID				:= fbJogCA.ErrorID;

jogca REF= stStatus;
END_METHOD

METHOD jogca_velo : REFERENCE TO stFeedback
VAR_INPUT
	bJogBackwards	: BOOL;
	bJogForward		: BOOL;
	lrVelocity		: LREAL;
END_VAR
VAR_INST
	stStatus		: stFeedback;
END_VAR
fbJogCA.JogBackwards			:= bJogBackwards;
fbJogCA.JogForward				:= bJogForward;
fbJogCA.Mode					:= E_JogMode.MC_JOGMODE_CONTINOUS;
fbJogCA.Velocity				:= lrVelocity;

stStatus.bDone					:= fbJogCA.Done;
stStatus.bBusy					:= fbJogCA.Busy;
stStatus.bCommandAborted		:= fbJogCA.CommandAborted;
stStatus.bError					:= fbJogCA.Error;
stStatus.udiErrorID				:= fbJogCA.ErrorID;

jogca_velo REF= stStatus;
END_METHOD

METHOD moveca : REFERENCE TO stFeedback
VAR_INPUT
	bExecute	: BOOL;
	lrPosition 	: LREAL;
	lrVelocity	: LREAL;
END_VAR
VAR_INST
	stStatus 	: stFeedback;
END_VAR
fbMoveAbsCA.Position 			:= lrPosition;
fbMoveAbsCA.Velocity			:= lrVelocity;
fbMoveAbsCA.Acceleration		:= stParameter.fAcceleration; 
fbMoveAbsCA.Deceleration		:= stParameter.fDeceleration; 
fbMoveAbsCA.Jerk				:= stParameter.fJerk; 
fbMoveAbsCA.Direction			:= tc3_mc3definitions.mcDirectionPositive;
fbMoveAbsCA.ContinuousUpdate 	:= TRUE;
fbMoveAbsCA.Execute				:= bExecute;
fbMoveAbsCA.Gap					:= MC_DEFAULT;
lrTargetPos 					:= lrPosition;

stStatus.bDone					:= fbMoveAbsCA.Done;
stStatus.bBusy					:= fbMoveAbsCA.Busy;
stStatus.bCommandAborted		:= fbMoveAbsCA.CommandAborted;
stStatus.bError					:= fbMoveAbsCA.Error;
stStatus.udiErrorID				:= fbMoveAbsCA.ErrorID;

moveca REF= stStatus;
END_METHOD

METHOD moveca_bytime : REFERENCE TO stFeedback
VAR_INPUT
	bExecute	: bool;
	lrPosition 	: LREAL;
	lrTime		: LREAL;
END_VAR
VAR_INST
	stStatus	: stFeedback;
END_VAR
fbMoveAbsTimeCA.bExecute 		:= bExecute;
fbMoveAbsTimeCA.lrPosition 		:= lrPosition;
fbMoveAbsTimeCA.lrTime			:= lrTime;
lrTargetPos 					:= lrPosition;

stStatus.bDone					:= fbMoveAbsTimeCA.Done;
stStatus.bBusy					:= fbMoveAbsTimeCA.Busy;
stStatus.bCommandAborted		:= fbMoveAbsTimeCA.CommandAborted;
stStatus.bError					:= fbMoveAbsTimeCA.Error;
stStatus.udiErrorID				:= fbMoveAbsTimeCA.ErrorID;

moveca_bytime REF= stStatus;
END_METHOD

METHOD moveca_direction : REFERENCE TO stFeedback
VAR_INPUT
	bExecute	: BOOL;
	lrPosition 	: LREAL;
	lrVelocity	: LREAL;
	Direction	: tc3_mc3definitions.MC_DIRECTION;
END_VAR
VAR_INST
	stStatus	: stFeedback;
END_VAR
fbMoveAbsCA.Position 			:= lrPosition;
fbMoveAbsCA.Velocity			:= lrVelocity;
fbMoveAbsCA.Acceleration		:= stParameter.fAcceleration; 
fbMoveAbsCA.Deceleration		:= stParameter.fDeceleration; 
fbMoveAbsCA.Jerk				:= stParameter.fJerk; 
fbMoveAbsCA.Direction			:= Direction;
fbMoveAbsCA.ContinuousUpdate 	:= TRUE;
fbMoveAbsCA.Execute				:= bExecute;
fbMoveAbsCA.Gap					:= MC_DEFAULT;
lrTargetPos 					:= lrPosition;

stStatus.bDone					:= fbMoveAbsCA.Done;
stStatus.bBusy					:= fbMoveAbsCA.Busy;
stStatus.bCommandAborted		:= fbMoveAbsCA.CommandAborted;
stStatus.bError					:= fbMoveAbsCA.Error;
stStatus.udiErrorID				:= fbMoveAbsCA.ErrorID;

moveca_direction REF= stStatus;
END_METHOD

METHOD moveca_gap : REFERENCE TO stFeedback
VAR_INPUT
	bExecute	: BOOL;
	lrPosition 	: LREAL;
	lrVelocity	: LREAL;
	lrGap		: LREAL;
END_VAR
VAR_INST
	stStatus	: stFeedback;
END_VAR
fbMoveAbsCA.Position 			:= lrPosition;
fbMoveAbsCA.Velocity			:= lrVelocity;
fbMoveAbsCA.Acceleration		:= stParameter.fAcceleration; 
fbMoveAbsCA.Deceleration		:= stParameter.fDeceleration; 
fbMoveAbsCA.Jerk				:= stParameter.fJerk; 
fbMoveAbsCA.Direction			:= tc3_mc3definitions.mcDirectionPositive;
fbMoveAbsCA.ContinuousUpdate 	:= TRUE;
fbMoveAbsCA.Execute				:= bExecute;
fbMoveAbsCA.Gap					:= lrGap;
lrTargetPos 					:= lrPosition;

stStatus.bDone					:= fbMoveAbsCA.Done;
stStatus.bBusy					:= fbMoveAbsCA.Busy;
stStatus.bCommandAborted		:= fbMoveAbsCA.CommandAborted;
stStatus.bError					:= fbMoveAbsCA.Error;
stStatus.udiErrorID				:= fbMoveAbsCA.ErrorID;

moveca_gap REF= stStatus;
END_METHOD

PROPERTY p_Axis : reference to AXIS_REF
GET
p_Axis ref= ax;
END_GET
SET
ax := p_Axis;
END_SET
END_PROPERTY

PROPERTY p_ModulePos : lreal
GET
p_ModulePos := ax.NcToPlc.ModuloActPos;
END_GET
END_PROPERTY

METHOD power_off : REFERENCE TO stFeedback
VAR_INST
	stStatus : stFeedback;
END_VAR
fbPower.Enable 			:= FALSE;
fbPower.Enable_Positive := FALSE;
fbPower.Enable_Negative := FALSE;
stStatus.bDone			:= NOT fbPower.Status;
stStatus.bBusy			:= fbPower.Busy;
stStatus.bError			:= fbPower.Error;
stStatus.udiErrorID		:= fbPower.ErrorID;
power_off 				REF= stStatus;
END_METHOD

METHOD power_on : REFERENCE TO stFeedback
VAR_INST
	stStatus : stFeedback;
END_VAR
fbPower.Enable 			:= TRUE;
fbPower.Enable_Positive := TRUE;
fbPower.Enable_Negative := TRUE;
stStatus.bDone			:= fbPower.Status;
stStatus.bBusy			:= fbPower.Busy;
stStatus.bError			:= fbPower.Error;
stStatus.udiErrorID		:= fbPower.ErrorID;
power_on 				REF= stStatus;
END_METHOD

METHOD reset : REFERENCE TO stFeedback
VAR_INPUT
	bExecute : BOOL;
END_VAR
VAR_INST
	stStatus : stFeedback;
END_VAR
fbReset.Execute			:= bExecute;
stStatus.bBusy			:= fbReset.Busy;
stStatus.bDone			:= fbReset.Done;
stStatus.bError			:= fbReset.Error;
stStatus.udiErrorID		:= fbReset.ErrorID;
reset REF= stStatus;
END_METHOD

METHOD standstill : BOOL
VAR_INPUT
END_VAR
standstill := ax.NcToPlc.SetVelo=0;
END_METHOD

END_FUNCTION_BLOCK

// ---- POUs/XTS/Movers/MC_MoveAbsoluteTimeCA.TcPOU
FUNCTION_BLOCK MC_MoveAbsoluteTimeCA 
VAR_IN_OUT
	Axis					: AXIS_REF; 
END_VAR
VAR_INPUT
	bExecute				: BOOL;
	lrPosition 				: LREAL;
	lrTime 					: LREAL;
END_VAR
VAR_OUTPUT
	Done					: BOOL;		 
	Busy 					: BOOL;
	Active					: BOOL;
	CommandAborted 			: BOOL;
	Error					: BOOL;
	ErrorId					: UDINT;	
END_VAR
VAR
	iState					: INT;
	lrDistance				: LREAL;
	fbReadParamSet			: MC_ReadParameterSet := (Execute := TRUE);
	stParameter				: ST_AxisParameterSet;
	fbMoveAbsoluteCA		: MC_MoveAbsoluteCA;
END_VAR

ReInit:
CASE iState OF
	
	0 : IF bExecute THEN iState := iState + 1; END_IF
	
	1 :
		fbReadParamSet(Parameter := stParameter, Axis := Axis, Execute := TRUE);
		IF fbReadParamSet.Done THEN
			iState := iState + 1;
			JMP ReInit; 
		END_IF
	2 :
		lrDistance := Tc2_Math.LMOD(lrPosition - axis.NcToPlc.ModuloSetPos + stParameter.fEncModuloFactor, stParameter.fEncModuloFactor);
		IF ABS(lrDistance) < 0.5 OR ABS(lrDistance-stParameter.fEncModuloFactor) < 0.5 THEN
			Done := TRUE;
			IF bExecute = FALSE THEN 
				fbMoveAbsoluteCA.Execute := FALSE;
				Done := FALSE;
				iState := 0; 
			END_IF
		ELSE 
			IF lrDistance < 0 THEN lrDistance := lrDistance + stParameter.fEncModuloFactor; END_IF
			fbMoveAbsoluteCA.Position		:= lrPosition;
			fbMoveAbsoluteCA.Velocity 		:= (lrDistance * 2.0) / lrTime;
			fbMoveAbsoluteCA.Acceleration 	:= (fbMoveAbsoluteCA.Velocity * 4.0) / lrTime;
			fbMoveAbsoluteCA.Deceleration 	:= (fbMoveAbsoluteCA.Velocity * 4.0) / lrTime;
			fbMoveAbsoluteCA.Jerk			:= (fbMoveAbsoluteCA.Acceleration * 4.0) / lrTime;
			fbMoveAbsoluteCA.Direction		:= tc3_mc3Definitions.MC_DIRECTION.mcDirectionPositive;
			iState := iState + 1;
			JMP ReInit;
		END_IF
		
	3 : //Execute
		fbMoveAbsoluteCA.Execute := TRUE;
		Done := fbMoveAbsoluteCA.Done;
		IF bExecute = FALSE THEN 
			fbMoveAbsoluteCA.Execute := FALSE;
			fbMoveAbsoluteCA(Axis:= Axis);
			Done := FALSE;
			iState := 0; 
			JMP ReInit;
		END_IF
	
END_CASE

fbMoveAbsoluteCA(
	Axis:= Axis, 
	Execute:= , 
	ContinuousUpdate:= , 
	Position:= , 
	Velocity:= , 
	Acceleration:= , 
	Deceleration:= , 
	Jerk:= , 
	Gap:= , 
	BufferMode:= , 
	Direction:= , 
	Options:= , 
	Done=> , 
	Busy=> Busy, 
	Active=> Active, 
	CommandAborted=> CommandAborted, 
	Error=> Error, 
	ErrorId=> ErrorId);

END_FUNCTION_BLOCK

// ---- POUs/XTS/Movers/MC_JogCA.TcPOU
FUNCTION_BLOCK MC_JogCA EXTENDS MC_Jog
VAR_INPUT
END_VAR
VAR_OUTPUT
END_VAR
VAR
	fbMoveRelativeCA 	: MC_MoveRelativeCA;
	fbHaltCA 			: MC_HaltCA;
	fbReadParameterSet	: MC_ReadParameterSet;
	stParameters		: st_axisparameterset;
	Old_bJogForward		: BOOL;
	Old_bJogBackwards	: BOOL;
	nState				: (IDLE, STARTING, EXECUTE, STOPPING, RESETING, ABORTED);
	bBackwards			: BOOL;
END_VAR


CASE nState OF
	
	IDLE://
		IF JogForward AND Old_bJogForward = FALSE THEN nState := RESETING; bBackwards := FALSE; Busy := TRUE; END_IF
		IF JogBackwards AND Old_bJogBackwards = FALSE THEN nState := RESETING; bBackwards := TRUE; Busy := TRUE; END_IF
		IF JogForward = FALSE AND JogBackwards = FALSE THEN Done := FALSE; END_IF
		
	RESETING:
		fbReadParameterSet(Parameter := stParameters, Axis := Axis, Execute := FALSE); 
		fbMoveRelativeCA(Axis := Axis, Execute := FALSE);	
		fbHaltCA(Axis := Axis, Execute := FALSE);
		nState := STARTING;
		
	STARTING:
	
		CASE Mode OF
			E_JogMode.MC_JOGMODE_CONTINOUS:
				fbReadParameterSet(Parameter := stParameters, Axis := Axis, Execute := TRUE, Error => Error, ErrorID => ErrorID); 
				fbMoveRelativeCA.Distance  	:= SEL(bBackwards, stParameters.fEncModuloFactor*100, -stParameters.fEncModuloFactor*100);
				fbMoveRelativeCA.Velocity	:= Velocity;
				IF fbReadParameterSet.Done THEN
					nState := EXECUTE;
				END_IF
				IF Error THEN nState := ABORTED; END_IF
			E_JogMode.MC_JOGMODE_INCHING:
        		//
			E_JogMode.MC_JOGMODE_INCHING_MODULO:  
        		//
			E_JogMode.MC_JOGMODE_STANDARD_FAST: 
				fbReadParameterSet(Parameter := stParameters, Axis := Axis, Execute := TRUE, Error => Error, ErrorID => ErrorID); 
				fbMoveRelativeCA.Distance  	:= SEL(bBackwards, stParameters.fEncModuloFactor*100, -stParameters.fEncModuloFactor*100);
				fbMoveRelativeCA.Velocity	:= stParameters.fVeloFastManual;
				IF fbReadParameterSet.Done THEN
					nState := EXECUTE;
				END_IF
				IF Error THEN nState := ABORTED; END_IF
			E_JogMode.MC_JOGMODE_STANDARD_SLOW:
				fbReadParameterSet(Parameter := stParameters, Axis := Axis, Execute := TRUE, Error => Error, ErrorID => ErrorID); 
				fbMoveRelativeCA.Distance  	:= SEL(bBackwards, stParameters.fEncModuloFactor*100, -stParameters.fEncModuloFactor*100);
				fbMoveRelativeCA.Velocity	:= stParameters.fVeloSlowManual;
				IF fbReadParameterSet.Done THEN
					nState := EXECUTE;
				END_IF
				IF Error THEN nState := ABORTED; END_IF
		END_CASE
		
	EXECUTE:

		fbMoveRelativeCA(Axis := Axis, Execute := TRUE, Active => Active, Error => Error, ErrorID => ErrorID, CommandAborted => CommandAborted, Done => Done);	
		IF (JogForward = FALSE AND bBackwards = FALSE) OR (JogBackwards = FALSE AND bBackwards = TRUE) THEN
			nState := STOPPING;
		END_IF
		IF Error THEN nState := ABORTED; END_IF
	
	STOPPING:
	
		fbHaltCA(Axis := Axis, Execute := TRUE, Error => Error, ErrorID => ErrorID, CommandAborted => CommandAborted, Done => Done);
		IF Error THEN nState := ABORTED; END_IF
		IF Done THEN nState := IDLE; Busy := FALSE; END_IF
		
	ABORTED:
		Active 	:= FALSE;
		Busy 	:= FALSE;
		Done	:= FALSE;
		IF (JogForward = FALSE AND bBackwards = FALSE) OR (JogBackwards = FALSE AND bBackwards = TRUE) THEN
			Error 	:= FALSE;
			nState 	:= IDLE;
		END_IF
	
END_CASE

Old_bJogForward := JogForward;

END_FUNCTION_BLOCK

// ---- POUs/XTS/Group CA/FB_GroupCA.TcPOU
FUNCTION_BLOCK FB_GroupCA EXTENDS FB_Mc2CaGroup
VAR_OUTPUT
	eGroupState			: MC_GROUP_STATE;
	bAllStandStill		: BOOL;
	bGroupError			: BOOL;
END_VAR
VAR 
	//Function Blocks
	ag					: AXES_GROUP_REF;
	fbEnable			: MC_GroupEnable;
	fbDisable			: MC_GroupDisable;
	fbHalt				: MC_GroupHalt;
	fbUnGroupAll		: MC_UngroupAllAxes;
	fbGroupStop			: MC_GroupStop;
	fbReset				: MC_GroupReset;
	fbState				: MC_GroupReadStatus;
	fbAddAxis2Group		: MC_AddAxisToGroup;
	
	uiSelectedMover		: UINT := 1;
	fbMovers			: REFERENCE TO ARRAY [1..Tc3_XTS_Utility.TcIoXtsEnvironmentParameterList.MaxXtsMoversPerXpu] OF FB_Mover;
	bInternalControl	: BOOL;
	bTmp				: BOOL;
END_VAR

METHOD clearcmd : BOOL
VAR_INPUT
END_VAR
halt(FALSE);
reset(FALSE);
ungroupall(FALSE);
enable(FALSE);
disable(FALSE);
END_METHOD

METHOD cyclic : BOOL
VAR_INPUT
	aMovers			: REFERENCE TO ARRAY [1..Tc3_XTS_Utility.TcIoXtsEnvironmentParameterList.MaxXtsMoversPerXpu] OF FB_Mover;
END_VAR
fbMovers REF= aMovers;

fbEnable(
	AxesGroup:= ag, 
	Execute:= , 
	Done=> , 
	Busy=> , 
	Error=> , 
	ErrorId=> );
	
fbDisable(
	AxesGroup:= ag, 
	Execute:= , 
	Done=> , 
	Busy=> , 
	Error=> , 
	ErrorId=> );
	
fbGroupStop(
	AxesGroup:= ag, 
	Execute:= , 
	Deceleration:= , 
	Jerk:= , 
	Done=> , 
	Busy=> , 
	Active=> , 
	CommandAborted=> , 
	Error=> , 
	ErrorId=> );
	
fbHalt(
	AxesGroup:= ag, 
	Execute:= , 
	Deceleration:= , 
	Jerk:= , 
	Done=> , 
	Busy=> , 
	Active=> , 
	CommandAborted=> , 
	Error=> , 
	ErrorId=> );
	
fbUnGroupAll(
	AxesGroup:= ag, 
	Execute:= , 
	Done=> , 
	Busy=> , 
	Error=> , 
	ErrorId=> );
	
fbReset(
	AxesGroup:= ag, 
	Execute:= , 
	Done=> , 
	Busy=> , 
	Error=> , 
	ErrorId=> );
	
fbState(
	AxesGroup:= ag, 
	Enable:= TRUE, 
	Valid=> , 
	Busy=> , 
	GroupMoving=> , 
	GroupHoming=> , 
	GroupErrorStop=> , 
	GroupNotReady=> , 
	GroupStandby=> , 
	GroupStopping=> , 
	GroupDisabled=> , 
	AllAxesStanding=> , 
	ConstantVelocity=> , 
	Accelerating=> , 
	Decelerating=> , 
	InPosition=> , 
	Error=> , 
	ErrorId=> );
	
IF __ISVALIDREF(fbMovers) THEN
	fbAddAxis2Group(
		AxesGroup:= ag, 
		Axis:= fbMovers[uiSelectedMover].p_Axis, 
		Execute:= , 
		IdentInGroup:= UDINT_TO_IDENTINGROUP(fbMovers[uiSelectedMover].udiID), 
		Done=> , 
		Busy=> , 
		Error=> , 
		ErrorId=> );
END_IF
	
IF fbState.GroupDisabled THEN
	eGroupState := MC_GROUP_STATE.mcGroupStateDisabled;
ELSIF fbState.GroupErrorStop THEN
	eGroupState := MC_GROUP_STATE.mcGroupStateErrorStop;
ELSIF fbState.GroupHoming THEN
	eGroupState := MC_GROUP_STATE.mcGroupStateHoming;
ELSIF fbState.GroupMoving THEN
	eGroupState := MC_GROUP_STATE.mcGroupStateMoving;
ELSIF fbState.GroupNotReady THEN
	eGroupState := MC_GROUP_STATE.mcGroupStateNotReady;
ELSIF fbState.GroupStandby THEN
	eGroupState := MC_GROUP_STATE.mcGroupStateStandby;
ELSIF fbState.GroupStopping THEN
	eGroupState := MC_GROUP_STATE.mcGroupStateStopping;
ELSIF fbState.GroupStandby THEN
	eGroupState := MC_GROUP_STATE.mcGroupStateSuspended;
ELSE
	eGroupState := MC_GROUP_STATE.mcGroupStateInvalid;
END_IF
bGroupError		 	:= eGroupState = mc_group_state.mcGroupStateErrorStop;
bAllStandStill 		:= fbState.AllAxesStanding;
END_METHOD

METHOD disable : REFERENCE TO stFeedback
VAR_INPUT
	bExecute : BOOL;
END_VAR
VAR_INST
	stStatus : stFeedback;
END_VAR
IF bInternalControl = FALSE THEN
	fbDisable.Execute 	:= bExecute;
	stStatus.bDone		:= fbDisable.Done;
	stStatus.bBusy		:= fbDisable.Busy;
	stStatus.bError		:= fbDisable.Error;
	stStatus.udiErrorID	:= fbDisable.ErrorId;
END_IF
disable REF= stStatus;
END_METHOD

METHOD enable : REFERENCE TO stFeedback 
VAR_INPUT
	bEnable : BOOL;
END_VAR
VAR_INST
	stStatus : stFeedback;
END_VAR
IF bInternalControl = FALSE THEN
	fbEnable.Execute 	:= bEnable;
	stStatus.bDone		:= fbEnable.Done;
	stStatus.bBusy		:= fbEnable.Busy;
	stStatus.bError		:= fbEnable.Error;
	stStatus.udiErrorID	:= fbEnable.ErrorId;
END_IF
enable REF= stStatus;
END_METHOD

METHOD halt : REFERENCE TO stFeedback
VAR_INPUT
	bExecute : BOOL;
END_VAR
VAR_INST
	stStatus : stFeedback;
END_VAR
IF bInternalControl = FALSE THEN
	fbHalt.Execute 		:= bExecute;
	stStatus.bDone		:= fbHalt.Done;
	stStatus.bBusy		:= fbHalt.Busy;
	stStatus.bError		:= fbHalt.Error;
	stStatus.udiErrorID	:= fbHalt.ErrorId;
END_IF
halt REF= stStatus;
END_METHOD

METHOD reset : REFERENCE TO stFeedback
VAR_INPUT
	bREset 		: BOOL;
END_VAR
VAR_INST
	stStatus : stFeedback;
END_VAR
IF bInternalControl = FALSE THEN
	fbReset.Execute 	:= bREset;
	stStatus.bDone		:= fbReset.Done;
	stStatus.bBusy		:= fbReset.Busy;
	stStatus.bError		:= fbReset.Error;
	stStatus.udiErrorID	:= fbReset.ErrorId;
END_IF
reset REF= stStatus;
END_METHOD

METHOD ungroupall : REFERENCE TO stFeedback
VAR_INPUT
	bExecute :BOOL;
END_VAR
VAR_INST
	stStatus : stFeedback;
END_VAR
IF bInternalControl = FALSE THEN
	fbUnGroupAll.Execute 	:= bExecute;
	stStatus.bDone			:= fbUnGroupAll.Done;
	stStatus.bBusy			:= fbUnGroupAll.Busy;
	stStatus.bError			:= fbUnGroupAll.Error;
	stStatus.udiErrorID		:= fbUnGroupAll.ErrorId;
END_IF
ungroupall REF= stStatus;
END_METHOD

END_FUNCTION_BLOCK

// ---- POUs/XTS/Stations/FB_Station.TcPOU
FUNCTION_BLOCK FB_Station EXTENDS FB_TcIoXtsInfoServerInfoStation
VAR
	ax						: REFERENCE TO ARRAY [1..Tc3_XTS_Utility.TcIoXtsEnvironmentParameterList.MaxXtsMoversPerXpu] OF FB_Mover;	//Movers
	stCfg 					: REFERENCE TO stStationCfg;
	udiNumMovers			: UDINT;		//Number of Movers into the system
	lrPartLength			: LREAL;
	bInvertPolarity			: BOOL;
	INextStation			: REFERENCE TO FB_Station;//I_Station;
END_VAR
VAR_OUTPUT
	udiNumMoversIn			: UDINT;		//Number of Movers into station
	udiErrorID				: UDINT;
END_VAR
VAR
	fbMoversFIFO			: FB_MoversFIFO;	
	bWaitingMovers			: BOOL;
	udiSequenceState		: UDINT;
	sMoversWaiting			: STRING;
	sMoversIn				: STRING;
	lrActualWaitingTime		: LREAL;
	lrActualProcessTime		: LREAL;
END_VAR
VAR
	bStart  				: BOOL;
	bStop					: BOOL;
	stSecuenceStatus		: stFeedback;
	bInternalControl		: bool;
END_VAR
VAR CONSTANT
	START_POSITION_ON_PART_STATION 	: DWORD := 16#03080272;
	END_POSITION_ON_PART_STATION 	: DWORD := 16#03080273;
	STOP_POSITIONS_STATION 			: DWORD := 16#0308028D;
END_VAR

PROPERTY Cfg : reference to stStationCfg
GET
Cfg REF= stCfg;
END_GET
END_PROPERTY

METHOD configure : BOOL
VAR_INPUT
	m_stCfg 				: REFERENCE TO stStationCfg;
	m_udiNumMovers			: UDINT;		//Number of Movers into the system
	m_lrPartLength			: LREAL;
	m_bInvertPolarity		: BOOL;
	m_INextStation			: REFERENCE TO FB_Station;//I_Station;
END_VAR
stCfg 			REF= m_stCfg 			;   
udiNumMovers	:= m_udiNumMovers		;  
lrPartLength	:= m_lrPartLength		;  
bInvertPolarity	:= m_bInvertPolarity	;
INextStation	ref= m_INextStation		;
END_METHOD

METHOD cyclic : BOOL
VAR_INPUT
	m_ax	: REFERENCE TO ARRAY [1..Tc3_XTS_Utility.TcIoXtsEnvironmentParameterList.MaxXtsMoversPerXpu] OF FB_Mover;
END_VAR
ax REF= m_ax;
fbMoversFIFO(ax := ax);	
stSecuenceStatus := MultipleStopSecuence(bStart, bStop);
END_METHOD

METHOD PRIVATE MultipleStopSecuence : REFERENCE TO stFeedback
VAR_INPUT
	bEnable 		: BOOL;
	bAbort			: BOOL;
END_VAR
VAR_INST
	udiState  			: UDINT;
	stCurrentCfg		: stStationCfg;
	fbTON				: ARRAY [1..5] OF TON;
	i					: UDINT;
	bAllDOne			: BOOL;
	m_bBusy				: BOOL;
	aMoversIN			: ARRAY [1..3] OF UDINT;
	ErrorID				: UDINT;
	tmInitProcessTime 	: TIME;
	tmInitWaitTime		: TIME;
	stStatus			: stFeedback;
END_VAR
(* 
	0. External Method to Add Movers into station
	1. Check if there is some mover in FIFO
	2. Send Mover to Stop Position
	3. Check Movers all StandStill and Reset Mover Commands
	4. Processing
	5. Send Movers to next FIFO Station
*)
IF bAbort AND udiState <> 100 THEN udiState := 100; END_IF

CASE udiState OF
	0 : //Wait for enable command
		IF bEnable THEN 
			udiNumMoversIn := 0;
			udiState := udiState + 10; 
		END_IF 
		
	10 : //Clear commands
		fbMoversFIFO.m_Clear();
		FOR i:=1 TO udiNumMovers DO
			//
			ax[i].clearCmd();
		END_FOR
		FOR i:= 1 TO 3 DO
			fbTon[i](IN := FALSE);
		END_FOR
		udiState := 19;
		
	19 : //Update configuration parameters
		stCurrentCfg 						:= stCfg;
		fbMoversFIFO.lrFirstStopPosition 	:= stCurrentCfg.lrStartPosition + stCurrentCfg.lrStopPosition[1];
		fbMoversFIFO.lrPartLength 			:= lrPartLength;
		tmInitWaitTime := TIME();
		udiState := udiState + 1;
		
	20 : //Check for new movers into FIFO
		m_bBusy 		:= TRUE;
		bWaitingMovers 	:= TRUE;
		IF fbMoversFIFO.nMovers > 0 AND udiNumMoversIn < stCurrentCfg.uiNumStopPositions THEN
			udiNumMoversIn 				:= udiNumMoversIn + 1;
			IF fbMoversFIFO.m_Extract(m_udiMoverID => aMoversIN[udiNumMoversIn]) THEN
				ax[aMoversIN[udiNumMoversIn]].clearCmd();
				bWaitingMovers := FALSE;
				udiState := udiState + 1;
			END_IF
		END_IF
		IF bEnable = FALSE THEN
			udiState := 100;
		END_IF
		
	21 : //Send Mover to Stop Position
		bAllDone := TRUE;
		FOR i:=1 TO udiNumMoversIn DO
			bAllDone := bAllDone AND ax[aMoversIN[i]].moveca_bytime(TRUE, stCurrentCfg.lrStartPosition + stCurrentCfg.lrStopPosition[stCurrentCfg.uiNumStopPositions - i + 1], stCfg.lrTravelTime).bDone;
			IF ax[aMoversIN[i]].moveca_bytime(TRUE, stCurrentCfg.lrStartPosition + stCurrentCfg.lrStopPosition[stCurrentCfg.uiNumStopPositions - i + 1], stCfg.lrTravelTime).bError THEN
				udiState := 999;
				EXIT;
			END_IF 
		END_FOR
		//If Station full process
		IF udiNumMoversIn = stCurrentCfg.uiNumStopPositions THEN
			IF bAllDone THEN 
				lrActualWaitingTime := (TIME_TO_LREAL(TIME() - tmInitWaitTime)-10.0)/1000.0;
				udiState := 30; 
			END_IF
		ELSE
			udiState := udiState - 1;
		END_IF
		
	30 : //Check if all movers are standstill and reset commands
		bAllDone := TRUE;
		FOR i:= 1 TO udiNumMoversIn DO	
			bAllDone := bAllDone AND ax[aMoversIN[i]].standstill();
			ax[aMoversIN[i]].clearCmd();
		END_FOR
		IF bAllDone THEN
			tmInitProcessTime := TIME();
			udiState := udiState + 10;
		END_IF
		
	40 : //Processing
		bAllDone := TRUE;
		FOR i:= 1 TO stCurrentCfg.uiNumStopPositions DO
			fbTon[i](IN := TRUE, PT := LREAL_TO_TIME(stCfg.lrProcessingTime*1000));
			bAllDone := bAllDone AND fbTON[i].Q;
		END_FOR
		IF (bAllDone AND stCfg.bEnableManualAck = FALSE) OR (stCfg.bEnableManualAck = TRUE AND stCfg.bManualAck) THEN
			FOR i:= 1 TO stCurrentCfg.uiNumStopPositions DO
				ax[aMoversIN[i]].clearCmd();
				fbTon[i](IN := FALSE);
			END_FOR
			lrActualProcessTime := (TIME_TO_LREAL(TIME() - tmInitProcessTime)-10.0)/1000.0;
			udiState := udiState + 10;
		END_IF
		
	50 : //Send out movers
		FOR i:= 1 TO udiNumMoversIn DO
		 	INextStation.RegisterMover(aMoversIN[i]);
			ax[aMoversIN[i]].moveca_bytime(TRUE, lrPosition := INextStation.Cfg.lrStartPosition, INextStation.Cfg.lrTravelTime);
		END_FOR
		udiNumMoversIn	:= 0;
		udiState 		:= 19;
		IF ErrorID <> 0 THEN
			udiState := 999;
		END_IF
		
	100 : //Abort
		m_bBusy := FALSE;
		bWaitingMovers := FALSE;
		IF bEnable = FALSE THEN
			ErrorID := 0;
			fbMoversFIFO.m_Clear();
			udiState := 0;
		END_IF
		
	999 : //Error
		m_bBusy := FALSE;
		bWaitingMovers := FALSE;
		IF bEnable = FALSE THEN
			fbMoversFIFO.m_Clear();
			ErrorID := 0;
			udiState := 0;
		END_IF
		
END_CASE
udiSequenceState 			:= udiState;
udiErrorID					:= ErrorID;
stStatus.udiErrorID			:= udiErrorID;
stStatus.bBusy				:= m_bBusy;
stStatus.bError				:= stStatus.udiErrorID <> 0;

MultipleStopSecuence		REF= stStatus;

sMoversWaiting := '';
FOR i:= 1 TO fbMoversFIFO.nMovers DO
	sMoversWaiting := CONCAT(sMoversWaiting, UDINT_TO_STRING(fbMoversFIFO.aMoversFIFO[i]));
	IF i < fbMoversFIFO.nMovers THEN sMoversWaiting := CONCAT(sMoversWaiting, ', '); END_IF
END_FOR
sMoversIn := '';
FOR i:= 1 TO udiNumMoversIn DO
	sMoversIn := CONCAT(sMoversIn, UDINT_TO_STRING(aMoversIN[i]));
	IF i < udiNumMoversIn THEN sMoversIn := concat(sMoversIn, ', '); END_IF
END_FOR
END_METHOD

METHOD RegisterMover : BOOL
VAR_INPUT
	udiMoverID : UDINT;
END_VAR
fbMoversFIFO.m_Add(udiMoverID);
END_METHOD

METHOD SetStationInfo : BOOL
VAR_INPUT
	bExecute		: BOOL;
	OTCID			: DWORD;
	bDisable		: BOOL;
END_VAR
VAR_INST
	iState 	 		: INT;
	fbADSWrite 		: adswrite;
	lrStartPos		: LREAL;
	lrEndPos		: LREAL;
	aStopPos		: ARRAY [1..3] OF LREAL;
	lrTmp			: LREAL;
	aTmp			: ARRAY [1..3] OF LREAL;
	lrDistance		: LREAL;
END_VAR

CASE iState OF
	0 : 
		IF bExecute THEN
			fbADSWrite(WRITE:= FALSE);
			fbMoversFIFO(ax := ax);	
			iState 	:= iState + 1;
		END_IF
	
	1 : //Write Init position
		lrStartPos 	:= SEL(bInvertPolarity, stCfg.lrStartPosition, lrPartLength - stCfg.lrEndPosition);
		lrEndPos 	:= SEL(bInvertPolarity, stCfg.lrEndPosition, lrPartLength - stCfg.lrStartPosition);
		IF bDisable THEN
			lrStartPos := lrEndPos := 0;
		END_IF
		fbADSWrite(
			NETID:= , 
			PORT:= 350, 
			IDXGRP:= OTCID, 
			IDXOFFS:= START_POSITION_ON_PART_STATION, 
			LEN:= SIZEOF(lrStartPos), 
			SRCADDR:= ADR(lrStartPos), 
			WRITE:= TRUE, 
			TMOUT:= , 
			BUSY=> , 
			ERR=> , 
			ERRID=> );
	
		IF fbADSWrite.BUSY = FALSE AND fbADSWrite.ERR = FALSE THEN
			fbADSWrite(WRITE := FALSE);
			iState := iState + 1;
		END_IF	
			
	2 : //Write End Position
		fbADSWrite(
			NETID:= , 
			PORT:= 350, 
			IDXGRP:= OTCID, 
			IDXOFFS:= END_POSITION_ON_PART_STATION, 
			LEN:= SIZEOF(lrEndPos), 
			SRCADDR:= ADR(lrEndPos), 
			WRITE:= TRUE, 
			TMOUT:= , 
			BUSY=> , 
			ERR=> , 
			ERRID=> );
	
		IF fbADSWrite.BUSY = FALSE AND fbADSWrite.ERR = FALSE THEN
			fbADSWrite(WRITE := FALSE);
			iState := iState + 1;
		END_IF
		
	3 : //Write Stop Positions
		aStopPos[1] := SEL(bInvertPolarity, stCfg.lrStopPosition[1], (stCfg.lrEndPosition - stCfg.lrStartPosition) - stCfg.lrStopPosition[1]); 
		aStopPos[2] := SEL(bInvertPolarity, stCfg.lrStopPosition[2], (stCfg.lrEndPosition - stCfg.lrStartPosition) - stCfg.lrStopPosition[2]); 
		aStopPos[3] := SEL(bInvertPolarity, stCfg.lrStopPosition[3], (stCfg.lrEndPosition - stCfg.lrStartPosition) - stCfg.lrStopPosition[3]); 
		IF stCfg.uiNumStopPositions = 1 AND NOT bDisable THEN
			aTmp[1] := aStopPos[1];
			aTmp[2] := aStopPos[1];
			aTmp[3] := aStopPos[1];
		ELSIF stCfg.uiNumStopPositions = 2 AND NOT bDisable THEN
			aTmp[1] := SEL(bInvertPolarity, aStopPos[1], aStopPos[2]);
			aTmp[2] := SEL(bInvertPolarity, aStopPos[2], aStopPos[1]);
			aTmp[3] := SEL(bInvertPolarity, aStopPos[2], aStopPos[1]);
		ELSIF stCfg.uiNumStopPositions = 3 AND NOT bDisable THEN
			aTmp[1] := SEL(bInvertPolarity, aStopPos[1], aStopPos[3]);
			aTmp[2] := SEL(bInvertPolarity, aStopPos[2], aStopPos[2]);
			aTmp[3] := SEL(bInvertPolarity, aStopPos[3], aStopPos[1]);
		ELSE
			aTmp[1]	:= 0.0;
			aTmp[2] := 0.0;
			aTmp[3] := 0.0;
		END_IF
		fbADSWrite(
			NETID:= , 
			PORT:= 350, 
			IDXGRP:= OTCID, 
			IDXOFFS:= STOP_POSITIONS_STATION, 
			LEN:= SIZEOF(aTmp), 
			SRCADDR:= ADR(aTmp), 
			WRITE:= TRUE, 
			TMOUT:= , 
			BUSY=> , 
			ERR=> , 
			ERRID=> );
	
		IF fbADSWrite.BUSY = FALSE AND fbADSWrite.ERR = FALSE THEN
			fbADSWrite(WRITE := FALSE);
			iState := iState + 1;
		END_IF
		
	4 : //Job Done
		SetStationInfo := TRUE;
		IF bExecute = FALSE THEN
			iState := 0;
		END_IF
	
END_CASE
END_METHOD

METHOD Start : BOOL
VAR_INPUT
END_VAR
bStart := TRUE;
bStop  := FALSE;
Start  := stSecuenceStatus.bBusy;
END_METHOD

METHOD Stop : BOOL
VAR_INPUT
END_VAR
bStart := FALSE;
bStop  := TRUE;
Stop   := NOT stSecuenceStatus.bBusy;
END_METHOD

END_FUNCTION_BLOCK

// ---- GlobalTextList.TcGTLO
TEXTLIST GlobalTextList
  991 = '     Done   Busy  Abort  Error         ErrorID'
  185 = '     Done   Busy  Abort  Error     ErrorID'
  381 = '     Done   Busy  CAborted     Error     ErrorID'
  98 = '    Coupled'
  946 = '    StandStill'
  454 = '  StandStill'
  73 = '%5.2f'
  853 = '%5.2f s/m'
  340 = '%d'
  70 = '%D'
  803 = '%i'
  164 = '%s'
  863 = '%x'
  1103 = '+'
  854 = '-'
  433 = 'Ack'
  784 = 'ActPos: %5.2f'
  935 = 'Actual Waiting Time'
  58 = 'ActVelo: %5.2f'
  772 = 'AllStandStill'
  436 = 'APPLY CONFIGURATION'
  210 = 'AUTO'
  154 = 'AUTOMATIC'
  2693 = 'Automatic'
  93 = 'Busy'
  147 = 'CONFIG'
  910 = 'CONFIGURATION'
  1010 = 'Configuration'
  142 = 'CONTROL'
  242 = 'Cycle Time'
  914 = 'Cycle Time: %5.2f s/mover'
  441 = 'DISABLE'
  194 = 'Distance between movers'
  402 = 'Done   Busy  CAborted     Error     ErrorID'
  405 = 'Done  Busy  CAborted     Error     ErrorID'
  49 = 'Done  Busy  CAborted  Error'
  844 = 'Done  Busy  CAborted  Error     ErrorID'
  992 = 'ENABLE'
  24 = 'Enable Visu Control, all methods will be locked'
  779 = 'Enabled'
  267 = 'End Position'
  860 = 'End Position: %5.2f'
  682 = 'End: %5.2f'
  605 = 'Error'
  443 = 'Error ID'
  174 = 'ErrorID: %i'
  183 = 'EXECUTE'
  933 = 'Execute      Done   Busy  CAborted     Error     ErrorID'
  529 = 'Extra Cfg.'
  961 = 'GROUP CA'
  823 = 'HALT'
  630 = 'HOME'
  360 = 'Id'
  214 = 'ID'
  2378 = 'Init Done'
  999 = 'Internal Control'
  677 = 'Invert Polarity'
  146 = 'JOG +'
  2714 = 'JOG -'
  309 = 'JOGGING'
  124 = 'Log: %s'
  215 = 'M. Ack'
  1878 = 'MANUAL'
  2735 = 'Manual'
  713 = 'Manual Ack'
  2444 = 'MOVE'
  228 = 'Mover ID: %d'
  45 = 'Mover mode'
  1070 = 'Mover Selection'
  973 = 'MOVER SELECTION'
  241 = 'MOVERS'
  696 = 'Movers In'
  923 = 'Movers In: %5.2f'
  1039 = 'Movers In: %s'
  902 = 'MOVERS SELECTION'
  286 = 'Movers Waiting'
  317 = 'Movers Waiting: %s'
  265 = 'Name'
  139 = 'Name: %5.2f'
  769 = 'Name: %s'
  235 = 'Not Configure Viewer'
  270 = 'Num Stop Positions'
  622 = 'Num Stop Positions: %d'
  686 = 'Number of Movers'
  958 = 'Number of Stations'
  503 = 'OPERATION'
  929 = 'POSITION'
  880 = 'Process Time'
  416 = 'Process Time: %5.2f'
  664 = 'Process Time: %5.2f s'
  272 = 'Process: %5.2f'
  301 = 'Process: %5.2f s'
  269 = 'Processing Time'
  176 = 'RESET'
  394 = 'RESULTS'
  899 = 'RUNTIME'
  679 = 'Runtime'
  208 = 'StandStill'
  1234 = 'START'
  266 = 'Start Position'
  240 = 'Start Position: %5.2f'
  408 = 'Start: %5.2f'
  813 = 'State'
  1046 = 'Station Selection'
  392 = 'STATION SELECTION'
  12 = 'STATIONS'
  570 = 'STATUS'
  771 = 'Status'
  724 = 'Status:'
  822 = 'Status: %D'
  42 = 'Status: %d'
  637 = 'Status: %s'
  437 = 'STOP'
  268 = 'Stop Position'
  634 = 'Stop Position 1: %5.2f'
  734 = 'Stop Position 2: %5.2f'
  934 = 'Stop Position 3: %5.2f'
  3040 = 'Stop Position Selection'
  112 = 'Stop Positions: %5.2f'
  904 = 'Stop Positions: %d'
  448 = 'Target Position'
  809 = 'Target Velocity'
  190 = 'TargetPos: %5.2f'
  579 = 'TEACH'
  3087 = 'TEACH STATION'
  271 = 'Travel Time'
  72 = 'Travel Time: %5.2f'
  261 = 'Waiting Time'
  950 = 'x'
END_TEXTLIST

// ---- POUs/XTS/Group CA/VI_GroupCAVisu.TcVIS
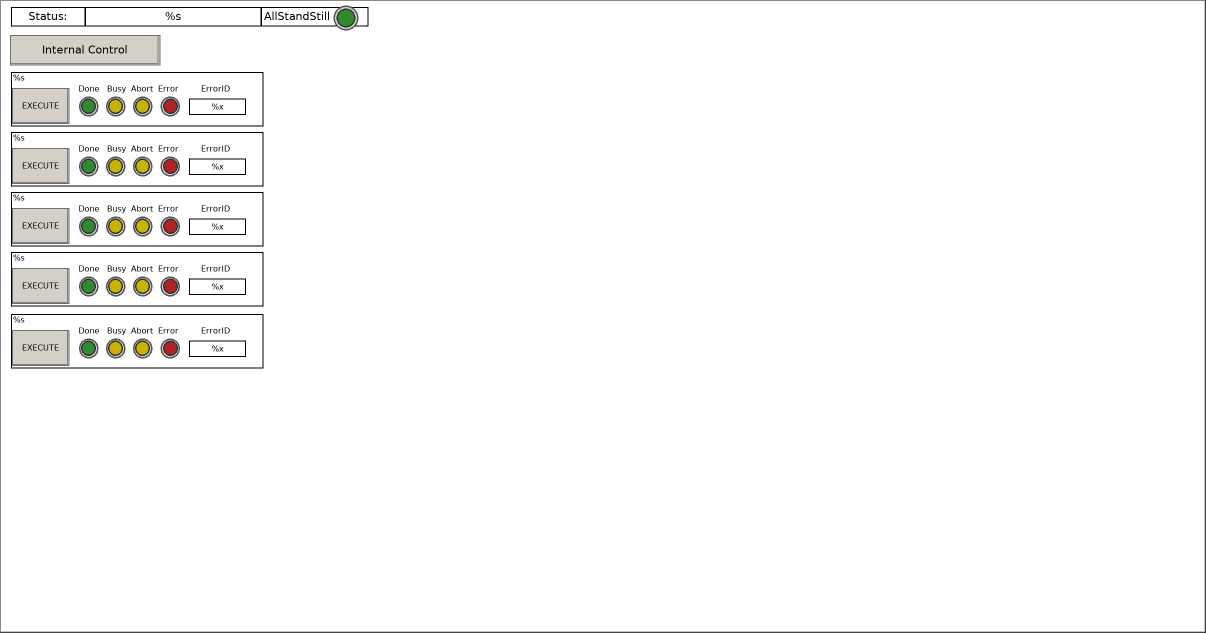
VISUALIZATION VI_GroupCAVisu  // 1206x633
VAR_IN_OUT
	gca : FB_GroupCA;
END_VAR
VAR
	stTableStruct : ARRAY [1..25] OF stTableStructx10;
END_VAR
    Rectangle (0,0 1206x633)
    Rectangle (85,7 176x19), "%s", text variable: gca.eGroupState, text list: 'GroupState_txt'
    Frame (11,72 252x54)
        shows VI_PLCOpenState(bExecute := gca.fbEnable.Execute, sName := 'Enable', bBusy := gca.fbEnable.Busy, bDone := gca.fbEnable.Done, bError := gca.fbEnable.Error, bCommandAborted := gca.bTmp, ErrorID := gca.fbEnable.ErrorId)
    Frame (11,132 252x54)
        shows VI_PLCOpenState(bExecute := gca.fbDisable.Execute, sName := 'Disable', bBusy := gca.fbDisable.Busy, bDone := gca.fbDisable.Done, bError := gca.fbDisable.Error, bCommandAborted := gca.bTmp, ErrorID := gca.fbDisable.ErrorId)
    Frame (11,192 252x54)
        shows VI_PLCOpenState(bExecute := gca.fbHalt.Execute, sName := 'Halt', bBusy := gca.fbHalt.Busy, bDone := gca.fbHalt.Done, bError := gca.fbHalt.Error, bCommandAborted := gca.fbHalt.CommandAborted, ErrorID := gca.fbHalt.ErrorId)
    Frame (11,252 252x54)
        shows VI_PLCOpenState(bExecute := gca.fbReset.Execute, sName := 'Reset', bBusy := gca.fbReset.Busy, bDone := gca.fbReset.Done, bError := gca.fbReset.Error, bCommandAborted := gca.bTmp, ErrorID := gca.fbReset.ErrorId)
    Rectangle (11,7 74x19), "Status:", text variable: gca.eGroupState
    Button (10,35 150x30), "Internal Control", tooltip "Enable Visu Control, all methods will be locked"
        toggle gca.bInternalControl
    Frame (11,314 252x54)
        shows VI_PLCOpenState(bExecute := gca.fbUnGroupAll.Execute, sName := 'UnGroupAll', bBusy := gca.fbUnGroupAll.Busy, bDone := gca.fbUnGroupAll.Done, bError := gca.fbUnGroupAll.Error, bCommandAborted := gca.bTmp, ErrorID := gca.fbUnGroupAll.ErrorId)
    Rectangle (261,7 107x19), "AllStandStill"
    Lamp1 (332,4 28x28), variable: gca.bAllStandStill, style: Lamp-Lamp1-Green
END_VISUALIZATION

